ACTION TEST_CASE_2_SETUP:
                        IF vTestCases[1].state = utTestCaseStates.ut_SETUP THEN
	(*Setup the test case information*)
	vTestCases[1].id := 2;
    vTestCases[1].desc[0] := 'RETURNS TRUE WHEN PARAMETER ACT EQUAL TO XP';
    vTestCases[1].desc[1] := 'Tests if the function returns True if the parameter act is equal to parameter xp';
	vTestCases[1].desc[2] := 'PASS IF: Return value is TRUE';
	
	(*Setup needed variables*)
	vTestCase2_act := REAL_TO_LREAL(115.4);
	vTestCase2_xp := REAL_TO_LREAL(115.4);
END_IF
                      
END_ACTION

ACTION TEST_CASE_2_EXEC:
                        IF vTestCases[1].state = utTestCaseStates.ut_RUNNING THEN
	(*Run the test case*)
	IF assertLessEqual_LREAL(vTestCase2_act, vTestCase2_xp) THEN
		vTestCases[1].state := utTestCaseStates.ut_PASSED;
		vTestCases[1].msg := 'Parameter act was equal to xp and function returned TRUE -> PASS';
	ELSE
		vTestCases[1].state := utTestCaseStates.ut_FAILED;
		vTestCases[1].msg := 'Parameter act was equal to xp and function returned FALSE -> FAIL';
	END_IF
END_IF
                      
END_ACTION
END_PROGRAM

PROGRAM test_assertArrayEqual_WORD
  VAR
    vTestCases : ARRAY[0..20] OF utTestCase;  (* Definition of all test cases for this POU *)
    testRunner : utTestSuite;  (* Test Suite fb instance to run the tests *)
    vRunAll : BOOL;  (* Manual command to run all tests for this POU *)
    vResetAll : BOOL;  (* Manual command to reset all tests for this POU *)
    vTestCase1_act : ARRAY[0..70] OF WORD;  (* Array data 1 of test case 1 *)
    vTestCase1_xp : ARRAY[0..70] OF WORD;  (* Array data 2 of test case 1 *)
    vTestCase2_act : ARRAY[0..70] OF WORD;  (* Array data 3 of test case 2 *)
    vTestCase2_xp : ARRAY[0..70] OF WORD;  (* Array data 4 of test case 2 *)
    i : UINT;  (* Iterator variable i *)
    j : UINT;  (* Iterator variable j *)
  END_VAR

                    (*Run the test cases*)
TEST_CASE_1_SETUP();
TEST_CASE_1_EXEC();

TEST_CASE_2_SETUP();
TEST_CASE_2_EXEC();

(*Instantiate the test runner*)
testRunner(
	Id := 140,
	Name := 'assertArrayEqual_WORD',
    RunTests := GVL.RunAll OR vRunAll,
	ResetTests := GVL.ResetAll OR vResetAll,
	TestCases:=vTestCases);

(*Report the results to the collection global*)
GVL.Results[testRunner.Id] := testRunner.Summary;
                  

ACTION TEST_CASE_1_SETUP:
                        IF vTestCases[0].state = utTestCaseStates.ut_SETUP THEN
	(*Setup the test case information*)
	vTestCases[0].id := 1;
	vTestCases[0].desc[0] := 'RETURNS TRUE WHEN ARRAYS EQUAL';
    vTestCases[0].desc[1] := 'Tests if the function returns True if the passed in arrays are identical';
	vTestCases[0].desc[2] := 'PASS IF: Return value is TRUE';
	
	(*Setup needed variables*)
	FOR i:=0 TO 70 DO
		vTestCase1_act[i] := UINT_TO_WORD(35 * BOOL_TO_UINT(i MOD 2 = 0));
		vTestCase1_xp[i] := UINT_TO_WORD(35 * BOOL_TO_UINT(i MOD 2 = 0));
	END_FOR
END_IF
                      
END_ACTION

ACTION TEST_CASE_1_EXEC:
                        IF vTestCases[0].state = utTestCaseStates.ut_RUNNING THEN
	(*Run the test case*)
	IF assertArrayEqual_WORD(ADR(vTestCase1_act), ADR(vTestCase1_xp), SIZEOF(vTestCase1_act)) THEN
		vTestCases[0].state := utTestCaseStates.ut_PASSED;
		vTestCases[0].msg := 'Arrays were equal and function returned TRUE -> PASS';
	ELSE
		vTestCases[0].state := utTestCaseStates.ut_FAILED;
		vTestCases[0].msg := 'Arrays were equal and function returned FALSE -> FAIL';
	END_IF
END_IF
                      
END_ACTION

ACTION TEST_CASE_2_SETUP:
                        IF vTestCases[1].state = utTestCaseStates.ut_SETUP THEN
	(*Setup the test case information*)
	vTestCases[1].id := 2;
	vTestCases[1].desc[0] := 'RETURNS FALSE WHEN ARRAYS NOT EQUAL';
    vTestCases[1].desc[1] := 'Tests if the function returns False if the passed in arrays are not identical';
	vTestCases[1].desc[2] := 'PASS IF: Return value is FALSE';
	
	(*Setup needed variables*)
	FOR j:=0 TO 70 DO
		vTestCase2_act[j] := UINT_TO_WORD(35 * BOOL_TO_UINT(j MOD 2 = 0));
		vTestCase2_xp[j] := UINT_TO_WORD(35 * BOOL_TO_UINT(j MOD 2 <> 0));
	END_FOR
END_IF
                      
END_ACTION

ACTION TEST_CASE_2_EXEC:
                        IF vTestCases[1].state = utTestCaseStates.ut_RUNNING THEN
	(*Run the test case*)
	IF NOT assertArrayEqual_WORD(ADR(vTestCase2_act), ADR(vTestCase2_xp), SIZEOF(vTestCase2_act)) THEN
		vTestCases[1].state := utTestCaseStates.ut_PASSED;
		vTestCases[1].msg := 'Arrays were not equal and function returned FALSE -> PASS';
	ELSE
		vTestCases[1].state := utTestCaseStates.ut_FAILED;
		vTestCases[1].msg := 'Arrays were not equal and function returned TRUE -> FAIL';
	END_IF
END_IF
                      
END_ACTION
END_PROGRAM

PROGRAM test_assertArrayEqual_DWORD
  VAR
    vTestCases : ARRAY[0..20] OF utTestCase;  (* Definition of all test cases for this POU *)
    testRunner : utTestSuite;  (* Test Suite fb instance to run the tests *)
    vRunAll : BOOL;  (* Manual command to run all tests for this POU *)
    vResetAll : BOOL;  (* Manual command to reset all tests for this POU *)
    vTestCase1_act : ARRAY[0..70] OF DWORD;  (* Array data 1 of test case 1 *)
    vTestCase1_xp : ARRAY[0..70] OF DWORD;  (* Array data 2 of test case 1 *)
    vTestCase2_act : ARRAY[0..70] OF DWORD;  (* Array data 3 of test case 2 *)
    vTestCase2_xp : ARRAY[0..70] OF DWORD;  (* Array data 4 of test case 2 *)
    i : UINT;  (* Iterator variable i *)
    j : UINT;  (* Iterator variable j *)
  END_VAR

                    (*Run the test cases*)
TEST_CASE_1_SETUP();
TEST_CASE_1_EXEC();

TEST_CASE_2_SETUP();
TEST_CASE_2_EXEC();

(*Instantiate the test runner*)
testRunner(
	Id := 141,
	Name := 'assertArrayEqual_DWORD',
    RunTests := GVL.RunAll OR vRunAll,
	ResetTests := GVL.ResetAll OR vResetAll,
	TestCases:=vTestCases);

(*Report the results to the collection global*)
GVL.Results[testRunner.Id] := testRunner.Summary;
                  

ACTION TEST_CASE_1_SETUP:
                        IF vTestCases[0].state = utTestCaseStates.ut_SETUP THEN
	(*Setup the test case information*)
	vTestCases[0].id := 1;
	vTestCases[0].desc[0] := 'RETURNS TRUE WHEN ARRAYS EQUAL';
    vTestCases[0].desc[1] := 'Tests if the function returns True if the passed in arrays are identical';
	vTestCases[0].desc[2] := 'PASS IF: Return value is TRUE';
	
	(*Setup needed variables*)
	FOR i:=0 TO 70 DO
		vTestCase1_act[i] := UINT_TO_DWORD(35 * BOOL_TO_UINT(i MOD 2 = 0));
		vTestCase1_xp[i] := UINT_TO_DWORD(35 * BOOL_TO_UINT(i MOD 2 = 0));
	END_FOR
END_IF
                      
END_ACTION

ACTION TEST_CASE_1_EXEC:
                        IF vTestCases[0].state = utTestCaseStates.ut_RUNNING THEN
	(*Run the test case*)
	IF assertArrayEqual_DWORD(ADR(vTestCase1_act), ADR(vTestCase1_xp), SIZEOF(vTestCase1_act)) THEN
		vTestCases[0].state := utTestCaseStates.ut_PASSED;
		vTestCases[0].msg := 'Arrays were equal and function returned TRUE -> PASS';
	ELSE
		vTestCases[0].state := utTestCaseStates.ut_FAILED;
		vTestCases[0].msg := 'Arrays were equal and function returned FALSE -> FAIL';
	END_IF
END_IF
                      
END_ACTION

ACTION TEST_CASE_2_SETUP:
                        IF vTestCases[1].state = utTestCaseStates.ut_SETUP THEN
	(*Setup the test case information*)
	vTestCases[1].id := 2;
	vTestCases[1].desc[0] := 'RETURNS FALSE WHEN ARRAYS NOT EQUAL';
    vTestCases[1].desc[1] := 'Tests if the function returns False if the passed in arrays are not identical';
	vTestCases[1].desc[2] := 'PASS IF: Return value is FALSE';
	
	(*Setup needed variables*)
	FOR j:=0 TO 70 DO
		vTestCase2_act[j] := UINT_TO_DWORD(35 * BOOL_TO_UINT(j MOD 2 = 0));
		vTestCase2_xp[j] := UINT_TO_DWORD(35 * BOOL_TO_UINT(j MOD 2 <> 0));
	END_FOR
END_IF
                      
END_ACTION

ACTION TEST_CASE_2_EXEC:
                        IF vTestCases[1].state = utTestCaseStates.ut_RUNNING THEN
	(*Run the test case*)
	IF NOT assertArrayEqual_DWORD(ADR(vTestCase2_act), ADR(vTestCase2_xp), SIZEOF(vTestCase2_act)) THEN
		vTestCases[1].state := utTestCaseStates.ut_PASSED;
		vTestCases[1].msg := 'Arrays were not equal and function returned FALSE -> PASS';
	ELSE
		vTestCases[1].state := utTestCaseStates.ut_FAILED;
		vTestCases[1].msg := 'Arrays were not equal and function returned TRUE -> FAIL';
	END_IF
END_IF
                      
END_ACTION
END_PROGRAM

PROGRAM test_assertArrayEqual_SINT
  VAR
    vTestCases : ARRAY[0..20] OF utTestCase;  (* Definition of all test cases for this POU *)
    testRunner : utTestSuite;  (* Test Suite fb instance to run the tests *)
    vRunAll : BOOL;  (* Manual command to run all tests for this POU *)
    vResetAll : BOOL;  (* Manual command to reset all tests for this POU *)
    vTestCase1_act : ARRAY[0..70] OF SINT;  (* Array data 1 of test case 1 *)
    vTestCase1_xp : ARRAY[0..70] OF SINT;  (* Array data 2 of test case 1 *)
    vTestCase2_act : ARRAY[0..70] OF SINT;  (* Array data 3 of test case 2 *)
    vTestCase2_xp : ARRAY[0..70] OF SINT;  (* Array data 4 of test case 2 *)
    i : UINT;  (* Iterator variable i *)
    j : UINT;  (* Iterator variable j *)
  END_VAR

                    (*Run the test cases*)
TEST_CASE_1_SETUP();
TEST_CASE_1_EXEC();

TEST_CASE_2_SETUP();
TEST_CASE_2_EXEC();

(*Instantiate the test runner*)
testRunner(
	Id := 143,
	Name := 'assertArrayEqual_SINT',
    RunTests := GVL.RunAll OR vRunAll,
	ResetTests := GVL.ResetAll OR vResetAll,
	TestCases:=vTestCases);

(*Report the results to the collection global*)
GVL.Results[testRunner.Id] := testRunner.Summary;
                  

ACTION TEST_CASE_1_SETUP:
                        IF vTestCases[0].state = utTestCaseStates.ut_SETUP THEN
	(*Setup the test case information*)
	vTestCases[0].id := 1;
	vTestCases[0].desc[0] := 'RETURNS TRUE WHEN ARRAYS EQUAL';
    vTestCases[0].desc[1] := 'Tests if the function returns True if the passed in arrays are identical';
	vTestCases[0].desc[2] := 'PASS IF: Return value is TRUE';
	
	(*Setup needed variables*)
	FOR i:=0 TO 70 DO
		vTestCase1_act[i] := UINT_TO_SINT(35 * BOOL_TO_UINT(i MOD 2 = 0));
		vTestCase1_xp[i] := UINT_TO_SINT(35 * BOOL_TO_UINT(i MOD 2 = 0));
	END_FOR
END_IF
                      
END_ACTION

ACTION TEST_CASE_1_EXEC:
                        IF vTestCases[0].state = utTestCaseStates.ut_RUNNING THEN
	(*Run the test case*)
	IF assertArrayEqual_SINT(ADR(vTestCase1_act), ADR(vTestCase1_xp), SIZEOF(vTestCase1_act)) THEN
		vTestCases[0].state := utTestCaseStates.ut_PASSED;
		vTestCases[0].msg := 'Arrays were equal and function returned TRUE -> PASS';
	ELSE
		vTestCases[0].state := utTestCaseStates.ut_FAILED;
		vTestCases[0].msg := 'Arrays were equal and function returned FALSE -> FAIL';
	END_IF
END_IF
                      
END_ACTION

ACTION TEST_CASE_2_SETUP:
                        IF vTestCases[1].state = utTestCaseStates.ut_SETUP THEN
	(*Setup the test case information*)
	vTestCases[1].id := 2;
	vTestCases[1].desc[0] := 'RETURNS FALSE WHEN ARRAYS NOT EQUAL';
    vTestCases[1].desc[1] := 'Tests if the function returns False if the passed in arrays are not identical';
	vTestCases[1].desc[2] := 'PASS IF: Return value is FALSE';
	
	(*Setup needed variables*)
	FOR j:=0 TO 70 DO
		vTestCase2_act[j] := UINT_TO_SINT(35 * BOOL_TO_UINT(j MOD 2 = 0));
		vTestCase2_xp[j] := UINT_TO_SINT(35 * BOOL_TO_UINT(j MOD 2 <> 0));
	END_FOR
END_IF
                      
END_ACTION

ACTION TEST_CASE_2_EXEC:
                        IF vTestCases[1].state = utTestCaseStates.ut_RUNNING THEN
	(*Run the test case*)
	IF NOT assertArrayEqual_SINT(ADR(vTestCase2_act), ADR(vTestCase2_xp), SIZEOF(vTestCase2_act)) THEN
		vTestCases[1].state := utTestCaseStates.ut_PASSED;
		vTestCases[1].msg := 'Arrays were not equal and function returned FALSE -> PASS';
	ELSE
		vTestCases[1].state := utTestCaseStates.ut_FAILED;
		vTestCases[1].msg := 'Arrays were not equal and function returned TRUE -> FAIL';
	END_IF
END_IF
                      
END_ACTION
END_PROGRAM

PROGRAM test_assertArrayEqual_LREAL
  VAR
    vTestCases : ARRAY[0..20] OF utTestCase;  (* Definition of all test cases for this POU *)
    testRunner : utTestSuite;  (* Test Suite fb instance to run the tests *)
    vRunAll : BOOL;  (* Manual command to run all tests for this POU *)
    vResetAll : BOOL;  (* Manual command to reset all tests for this POU *)
    vTestCase1_act : ARRAY[0..70] OF LREAL;  (* Array data 1 of test case 1 *)
    vTestCase1_xp : ARRAY[0..70] OF LREAL;  (* Array data 2 of test case 1 *)
    vTestCase2_act : ARRAY[0..70] OF LREAL;  (* Array data 3 of test case 2 *)
    vTestCase2_xp : ARRAY[0..70] OF LREAL;  (* Array data 4 of test case 2 *)
    i : UINT;  (* Iterator variable i *)
    j : UINT;  (* Iterator variable j *)
  END_VAR

                    (*Run the test cases*)
TEST_CASE_1_SETUP();
TEST_CASE_1_EXEC();

TEST_CASE_2_SETUP();
TEST_CASE_2_EXEC();

(*Instantiate the test runner*)
testRunner(
	Id := 152,
	Name := 'assertArrayEqual_LREAL',
    RunTests := GVL.RunAll OR vRunAll,
	ResetTests := GVL.ResetAll OR vResetAll,
	TestCases:=vTestCases);

(*Report the results to the collection global*)
GVL.Results[testRunner.Id] := testRunner.Summary;
                  

ACTION TEST_CASE_1_EXEC:
                        IF vTestCases[0].state = utTestCaseStates.ut_RUNNING THEN
	(*Run the test case*)
	IF assertArrayEqual_LREAL(ADR(vTestCase1_act), ADR(vTestCase1_xp), SIZEOF(vTestCase1_act)) THEN
		vTestCases[0].state := utTestCaseStates.ut_PASSED;
		vTestCases[0].msg := 'Arrays were equal and function returned TRUE -> PASS';
	ELSE
		vTestCases[0].state := utTestCaseStates.ut_FAILED;
		vTestCases[0].msg := 'Arrays were equal and function returned FALSE -> FAIL';
	END_IF
END_IF
                      
END_ACTION

ACTION TEST_CASE_2_SETUP:
                        IF vTestCases[1].state = utTestCaseStates.ut_SETUP THEN
	(*Setup the test case information*)
	vTestCases[1].id := 2;
	vTestCases[1].desc[0] := 'RETURNS FALSE WHEN ARRAYS NOT EQUAL';
    vTestCases[1].desc[1] := 'Tests if the function returns False if the passed in arrays are not identical';
	vTestCases[1].desc[2] := 'PASS IF: Return value is FALSE';
	
	(*Setup needed variables*)
	FOR j:=0 TO 70 DO
		vTestCase2_act[j] := UINT_TO_LREAL(35 * BOOL_TO_UINT(j MOD 2 = 0));
		vTestCase2_xp[j] := UINT_TO_LREAL(35 * BOOL_TO_UINT(j MOD 2 <> 0));
	END_FOR
END_IF
                      
END_ACTION

ACTION TEST_CASE_2_EXEC:
                        IF vTestCases[1].state = utTestCaseStates.ut_RUNNING THEN
	(*Run the test case*)
	IF NOT assertArrayEqual_LREAL(ADR(vTestCase2_act), ADR(vTestCase2_xp), SIZEOF(vTestCase2_act)) THEN
		vTestCases[1].state := utTestCaseStates.ut_PASSED;
		vTestCases[1].msg := 'Arrays were not equal and function returned FALSE -> PASS';
	ELSE
		vTestCases[1].state := utTestCaseStates.ut_FAILED;
		vTestCases[1].msg := 'Arrays were not equal and function returned TRUE -> FAIL';
	END_IF
END_IF
                      
END_ACTION

ACTION TEST_CASE_1_SETUP:
                        IF vTestCases[0].state = utTestCaseStates.ut_SETUP THEN
	(*Setup the test case information*)
	vTestCases[0].id := 1;
	vTestCases[0].desc[0] := 'RETURNS TRUE WHEN ARRAYS EQUAL';
    vTestCases[0].desc[1] := 'Tests if the function returns True if the passed in arrays are identical';
	vTestCases[0].desc[2] := 'PASS IF: Return value is TRUE';
	
	(*Setup needed variables*)
	FOR i:=0 TO 70 DO
		vTestCase1_act[i] := UINT_TO_LREAL(35 * BOOL_TO_UINT(i MOD 2 = 0));
		vTestCase1_xp[i] := UINT_TO_LREAL(35 * BOOL_TO_UINT(i MOD 2 = 0));
	END_FOR
END_IF
                      
END_ACTION
END_PROGRAM

PROGRAM test_assertLessEqual_LTIME
  VAR
    vTestCases : ARRAY[0..20] OF utTestCase;  (* Definition of all test cases for this POU *)
    testRunner : utTestSuite;  (* Test Suite fb instance to run the tests *)
    vRunAll : BOOL;  (* Manual command to run all tests for this POU *)
    vResetAll : BOOL;  (* Manual command to reset all tests for this POU *)
    vTestCase1_act : LTIME;  (* Test data 1 of test case 1 *)
    vTestCase1_xp : LTIME;  (* Test data 2 of test case 1 *)
    vTestCase2_act : LTIME;  (* Test data 1 of test case 2 *)
    vTestCase2_xp : LTIME;  (* Test data 2 of test case 2 *)
    vTestCase3_act : LTIME;  (* Test data 1 of test case 3 *)
    vTestCase3_xp : LTIME;  (* Test data 2 of test case 3 *)
  END_VAR

                    (*Run the test cases*)
TEST_CASE_1_SETUP();
TEST_CASE_1_EXEC();

TEST_CASE_2_SETUP();
TEST_CASE_2_EXEC();

TEST_CASE_3_SETUP();
TEST_CASE_3_EXEC();

(*Instantiate the test runner*)
testRunner(
	Id := 131,
	Name := 'assertLessEqual_LTIME',
    RunTests := GVL.RunAll OR vRunAll,
	ResetTests := GVL.ResetAll OR vResetAll,
	TestCases:=vTestCases);

(*Report the results to the collection global*)
GVL.Results[testRunner.Id] := testRunner.Summary;
                  

ACTION TEST_CASE_1_EXEC:
                        IF vTestCases[0].state = utTestCaseStates.ut_RUNNING THEN
	(*Run the test case*)
	IF assertLessEqual_LTIME(vTestCase1_act, vTestCase1_xp) THEN
		vTestCases[0].state := utTestCaseStates.ut_PASSED;
		vTestCases[0].msg := 'Parameter act was less than xp and function returned TRUE -> PASS';
	ELSE
		vTestCases[0].state := utTestCaseStates.ut_FAILED;
		vTestCases[0].msg := 'Parameter act was less than xp and function returned FALSE -> FAIL';
	END_IF
END_IF
                      
END_ACTION

ACTION TEST_CASE_3_SETUP:
                        IF vTestCases[2].state = utTestCaseStates.ut_SETUP THEN
	(*Setup the test case information*)
	vTestCases[2].id := 3;
    vTestCases[2].desc[0] := 'RETURNS FALSE WHEN PARAMETER ACT GREATER THAN XP';
    vTestCases[2].desc[1] := 'Tests if the function returns False if the parameter act is greater than parameter xp';
	vTestCases[2].desc[2] := 'PASS IF: Return value is FALSE';
	
	(*Setup needed variables*)
	vTestCase3_act := REAL_TO_LTIME(115.4);
	vTestCase3_xp := REAL_TO_LTIME(85.4);
END_IF
                      
END_ACTION

ACTION TEST_CASE_3_EXEC:
                        IF vTestCases[2].state = utTestCaseStates.ut_RUNNING THEN
	(*Run the test case*)
	IF NOT assertLessEqual_LTIME(vTestCase3_act, vTestCase3_xp) THEN
		vTestCases[2].state := utTestCaseStates.ut_PASSED;
		vTestCases[2].msg := 'Parameter act was greater than xp and function returned FALSE -> PASS';
	ELSE
		vTestCases[2].state := utTestCaseStates.ut_FAILED;
		vTestCases[2].msg := 'Parameter act was greater than xp and function returned TRUE -> FAIL';
	END_IF
END_IF
                      
END_ACTION

ACTION TEST_CASE_1_SETUP:
                        IF vTestCases[0].state = utTestCaseStates.ut_SETUP THEN
	(*Setup the test case information*)
	vTestCases[0].id := 1;
	vTestCases[0].desc[0] := 'RETURNS TRUE WHEN PARAMETER ACT LESS THAN XP';
    vTestCases[0].desc[1] := 'Tests if the function returns True if the parameter act is less than parameter xp';
	vTestCases[0].desc[2] := 'PASS IF: Return value is TRUE';
	
	(*Setup needed variables*)
	vTestCase1_act := REAL_TO_LTIME(85.4);
	vTestCase1_xp := REAL_TO_LTIME(115.4);
END_IF
                      
END_ACTION

ACTION TEST_CASE_2_SETUP:
                        IF vTestCases[1].state = utTestCaseStates.ut_SETUP THEN
	(*Setup the test case information*)
	vTestCases[1].id := 2;
    vTestCases[1].desc[0] := 'RETURNS TRUE WHEN PARAMETER ACT EQUAL TO XP';
    vTestCases[1].desc[1] := 'Tests if the function returns True if the parameter act is equal to parameter xp';
	vTestCases[1].desc[2] := 'PASS IF: Return value is TRUE';
	
	(*Setup needed variables*)
	vTestCase2_act := REAL_TO_LTIME(115.4);
	vTestCase2_xp := REAL_TO_LTIME(115.4);
END_IF
                      
END_ACTION

ACTION TEST_CASE_2_EXEC:
                        IF vTestCases[1].state = utTestCaseStates.ut_RUNNING THEN
	(*Run the test case*)
	IF assertLessEqual_LTIME(vTestCase2_act, vTestCase2_xp) THEN
		vTestCases[1].state := utTestCaseStates.ut_PASSED;
		vTestCases[1].msg := 'Parameter act was equal to xp and function returned TRUE -> PASS';
	ELSE
		vTestCases[1].state := utTestCaseStates.ut_FAILED;
		vTestCases[1].msg := 'Parameter act was equal to xp and function returned FALSE -> FAIL';
	END_IF
END_IF
                      
END_ACTION
END_PROGRAM

PROGRAM test_assertArrayEqual_LINT
  VAR
    vTestCases : ARRAY[0..20] OF utTestCase;  (* Definition of all test cases for this POU *)
    testRunner : utTestSuite;  (* Test Suite fb instance to run the tests *)
    vRunAll : BOOL;  (* Manual command to run all tests for this POU *)
    vResetAll : BOOL;  (* Manual command to reset all tests for this POU *)
    vTestCase1_act : ARRAY[0..70] OF LINT;  (* Array data 1 of test case 1 *)
    vTestCase1_xp : ARRAY[0..70] OF LINT;  (* Array data 2 of test case 1 *)
    vTestCase2_act : ARRAY[0..70] OF LINT;  (* Array data 3 of test case 2 *)
    vTestCase2_xp : ARRAY[0..70] OF LINT;  (* Array data 4 of test case 2 *)
    i : UINT;  (* Iterator variable i *)
    j : UINT;  (* Iterator variable j *)
  END_VAR

                    (*Run the test cases*)
TEST_CASE_1_SETUP();
TEST_CASE_1_EXEC();

TEST_CASE_2_SETUP();
TEST_CASE_2_EXEC();

(*Instantiate the test runner*)
testRunner(
	Id := 149,
	Name := 'assertArrayEqual_LINT',
    RunTests := GVL.RunAll OR vRunAll,
	ResetTests := GVL.ResetAll OR vResetAll,
	TestCases:=vTestCases);

(*Report the results to the collection global*)
GVL.Results[testRunner.Id] := testRunner.Summary;
                  

ACTION TEST_CASE_2_SETUP:
                        IF vTestCases[1].state = utTestCaseStates.ut_SETUP THEN
	(*Setup the test case information*)
	vTestCases[1].id := 2;
	vTestCases[1].desc[0] := 'RETURNS FALSE WHEN ARRAYS NOT EQUAL';
    vTestCases[1].desc[1] := 'Tests if the function returns False if the passed in arrays are not identical';
	vTestCases[1].desc[2] := 'PASS IF: Return value is FALSE';
	
	(*Setup needed variables*)
	FOR j:=0 TO 70 DO
		vTestCase2_act[j] := UINT_TO_LINT(35 * BOOL_TO_UINT(j MOD 2 = 0));
		vTestCase2_xp[j] := UINT_TO_LINT(35 * BOOL_TO_UINT(j MOD 2 <> 0));
	END_FOR
END_IF
                      
END_ACTION

ACTION TEST_CASE_1_SETUP:
                        IF vTestCases[0].state = utTestCaseStates.ut_SETUP THEN
	(*Setup the test case information*)
	vTestCases[0].id := 1;
	vTestCases[0].desc[0] := 'RETURNS TRUE WHEN ARRAYS EQUAL';
    vTestCases[0].desc[1] := 'Tests if the function returns True if the passed in arrays are identical';
	vTestCases[0].desc[2] := 'PASS IF: Return value is TRUE';
	
	(*Setup needed variables*)
	FOR i:=0 TO 70 DO
		vTestCase1_act[i] := UINT_TO_LINT(35 * BOOL_TO_UINT(i MOD 2 = 0));
		vTestCase1_xp[i] := UINT_TO_LINT(35 * BOOL_TO_UINT(i MOD 2 = 0));
	END_FOR
END_IF
                      
END_ACTION

ACTION TEST_CASE_1_EXEC:
                        IF vTestCases[0].state = utTestCaseStates.ut_RUNNING THEN
	(*Run the test case*)
	IF assertArrayEqual_LINT(ADR(vTestCase1_act), ADR(vTestCase1_xp), SIZEOF(vTestCase1_act)) THEN
		vTestCases[0].state := utTestCaseStates.ut_PASSED;
		vTestCases[0].msg := 'Arrays were equal and function returned TRUE -> PASS';
	ELSE
		vTestCases[0].state := utTestCaseStates.ut_FAILED;
		vTestCases[0].msg := 'Arrays were equal and function returned FALSE -> FAIL';
	END_IF
END_IF
                      
END_ACTION

ACTION TEST_CASE_2_EXEC:
                        IF vTestCases[1].state = utTestCaseStates.ut_RUNNING THEN
	(*Run the test case*)
	IF NOT assertArrayEqual_LINT(ADR(vTestCase2_act), ADR(vTestCase2_xp), SIZEOF(vTestCase2_act)) THEN
		vTestCases[1].state := utTestCaseStates.ut_PASSED;
		vTestCases[1].msg := 'Arrays were not equal and function returned FALSE -> PASS';
	ELSE
		vTestCases[1].state := utTestCaseStates.ut_FAILED;
		vTestCases[1].msg := 'Arrays were not equal and function returned TRUE -> FAIL';
	END_IF
END_IF
                      
END_ACTION
END_PROGRAM

PROGRAM test_assertLessEqual_REAL
  VAR
    vTestCases : ARRAY[0..20] OF utTestCase;  (* Definition of all test cases for this POU *)
    testRunner : utTestSuite;  (* Test Suite fb instance to run the tests *)
    vRunAll : BOOL;  (* Manual command to run all tests for this POU *)
    vResetAll : BOOL;  (* Manual command to reset all tests for this POU *)
    vTestCase1_act : REAL;  (* Test data 1 of test case 1 *)
    vTestCase1_xp : REAL;  (* Test data 2 of test case 1 *)
    vTestCase2_act : REAL;  (* Test data 1 of test case 2 *)
    vTestCase2_xp : REAL;  (* Test data 2 of test case 2 *)
    vTestCase3_act : REAL;  (* Test data 1 of test case 3 *)
    vTestCase3_xp : REAL;  (* Test data 2 of test case 3 *)
  END_VAR

                    (*Run the test cases*)
TEST_CASE_1_SETUP();
TEST_CASE_1_EXEC();

TEST_CASE_2_SETUP();
TEST_CASE_2_EXEC();

TEST_CASE_3_SETUP();
TEST_CASE_3_EXEC();

(*Instantiate the test runner*)
testRunner(
	Id := 128,
	Name := 'assertLessEqual_REAL',
    RunTests := GVL.RunAll OR vRunAll,
	ResetTests := GVL.ResetAll OR vResetAll,
	TestCases:=vTestCases);

(*Report the results to the collection global*)
GVL.Results[testRunner.Id] := testRunner.Summary;
                  

ACTION TEST_CASE_2_SETUP:
                        IF vTestCases[1].state = utTestCaseStates.ut_SETUP THEN
	(*Setup the test case information*)
	vTestCases[1].id := 2;
    vTestCases[1].desc[0] := 'RETURNS TRUE WHEN PARAMETER ACT EQUAL TO XP';
    vTestCases[1].desc[1] := 'Tests if the function returns True if the parameter act is equal to parameter xp';
	vTestCases[1].desc[2] := 'PASS IF: Return value is TRUE';
	
	(*Setup needed variables*)
	vTestCase2_act := 115.4;
	vTestCase2_xp := 115.4;
END_IF
                      
END_ACTION

ACTION TEST_CASE_3_SETUP:
                        IF vTestCases[2].state = utTestCaseStates.ut_SETUP THEN
	(*Setup the test case information*)
	vTestCases[2].id := 3;
    vTestCases[2].desc[0] := 'RETURNS FALSE WHEN PARAMETER ACT GREATER THAN XP';
    vTestCases[2].desc[1] := 'Tests if the function returns False if the parameter act is greater than parameter xp';
	vTestCases[2].desc[2] := 'PASS IF: Return value is FALSE';
	
	(*Setup needed variables*)
	vTestCase3_act := 115.4;
	vTestCase3_xp := 85.4;
END_IF
                      
END_ACTION

ACTION TEST_CASE_3_EXEC:
                        IF vTestCases[2].state = utTestCaseStates.ut_RUNNING THEN
	(*Run the test case*)
	IF NOT assertLessEqual_REAL(vTestCase3_act, vTestCase3_xp) THEN
		vTestCases[2].state := utTestCaseStates.ut_PASSED;
		vTestCases[2].msg := 'Parameter act was greater than xp and function returned FALSE -> PASS';
	ELSE
		vTestCases[2].state := utTestCaseStates.ut_FAILED;
		vTestCases[2].msg := 'Parameter act was greater than xp and function returned TRUE -> FAIL';
	END_IF
END_IF
                      
END_ACTION

ACTION TEST_CASE_2_EXEC:
                        IF vTestCases[1].state = utTestCaseStates.ut_RUNNING THEN
	(*Run the test case*)
	IF assertLessEqual_REAL(vTestCase2_act, vTestCase2_xp) THEN
		vTestCases[1].state := utTestCaseStates.ut_PASSED;
		vTestCases[1].msg := 'Parameter act was equal to xp and function returned TRUE -> PASS';
	ELSE
		vTestCases[1].state := utTestCaseStates.ut_FAILED;
		vTestCases[1].msg := 'Parameter act was equal to xp and function returned FALSE -> FAIL';
	END_IF
END_IF
                      
END_ACTION

ACTION TEST_CASE_1_SETUP:
                        IF vTestCases[0].state = utTestCaseStates.ut_SETUP THEN
	(*Setup the test case information*)
	vTestCases[0].id := 1;
	vTestCases[0].desc[0] := 'RETURNS TRUE WHEN PARAMETER ACT LESS THAN XP';
    vTestCases[0].desc[1] := 'Tests if the function returns True if the parameter act is less than parameter xp';
	vTestCases[0].desc[2] := 'PASS IF: Return value is TRUE';
	
	(*Setup needed variables*)
	vTestCase1_act := 85.4;
	vTestCase1_xp := 115.4;
END_IF
                      
END_ACTION

ACTION TEST_CASE_1_EXEC:
                        IF vTestCases[0].state = utTestCaseStates.ut_RUNNING THEN
	(*Run the test case*)
	IF assertLessEqual_REAL(vTestCase1_act, vTestCase1_xp) THEN
		vTestCases[0].state := utTestCaseStates.ut_PASSED;
		vTestCases[0].msg := 'Parameter act was less than xp and function returned TRUE -> PASS';
	ELSE
		vTestCases[0].state := utTestCaseStates.ut_FAILED;
		vTestCases[0].msg := 'Parameter act was less than xp and function returned FALSE -> FAIL';
	END_IF
END_IF
                      
END_ACTION
END_PROGRAM

PROGRAM test_assertArrayEqual_DINT
  VAR
    vTestCases : ARRAY[0..20] OF utTestCase;  (* Definition of all test cases for this POU *)
    testRunner : utTestSuite;  (* Test Suite fb instance to run the tests *)
    vRunAll : BOOL;  (* Manual command to run all tests for this POU *)
    vResetAll : BOOL;  (* Manual command to reset all tests for this POU *)
    vTestCase1_act : ARRAY[0..70] OF DINT;  (* Array data 1 of test case 1 *)
    vTestCase1_xp : ARRAY[0..70] OF DINT;  (* Array data 2 of test case 1 *)
    vTestCase2_act : ARRAY[0..70] OF DINT;  (* Array data 3 of test case 2 *)
    vTestCase2_xp : ARRAY[0..70] OF DINT;  (* Array data 4 of test case 2 *)
    i : UINT;  (* Iterator variable i *)
    j : UINT;  (* Iterator variable j *)
  END_VAR

                    (*Run the test cases*)
TEST_CASE_1_SETUP();
TEST_CASE_1_EXEC();

TEST_CASE_2_SETUP();
TEST_CASE_2_EXEC();

(*Instantiate the test runner*)
testRunner(
	Id := 147,
	Name := 'assertArrayEqual_DINT',
    RunTests := GVL.RunAll OR vRunAll,
	ResetTests := GVL.ResetAll OR vResetAll,
	TestCases:=vTestCases);

(*Report the results to the collection global*)
GVL.Results[testRunner.Id] := testRunner.Summary;
                  

ACTION TEST_CASE_1_SETUP:
                        IF vTestCases[0].state = utTestCaseStates.ut_SETUP THEN
	(*Setup the test case information*)
	vTestCases[0].id := 1;
	vTestCases[0].desc[0] := 'RETURNS TRUE WHEN ARRAYS EQUAL';
    vTestCases[0].desc[1] := 'Tests if the function returns True if the passed in arrays are identical';
	vTestCases[0].desc[2] := 'PASS IF: Return value is TRUE';
	
	(*Setup needed variables*)
	FOR i:=0 TO 70 DO
		vTestCase1_act[i] := UINT_TO_DINT(35 * BOOL_TO_UINT(i MOD 2 = 0));
		vTestCase1_xp[i] := UINT_TO_DINT(35 * BOOL_TO_UINT(i MOD 2 = 0));
	END_FOR
END_IF
                      
END_ACTION

ACTION TEST_CASE_1_EXEC:
                        IF vTestCases[0].state = utTestCaseStates.ut_RUNNING THEN
	(*Run the test case*)
	IF assertArrayEqual_DINT(ADR(vTestCase1_act), ADR(vTestCase1_xp), SIZEOF(vTestCase1_act)) THEN
		vTestCases[0].state := utTestCaseStates.ut_PASSED;
		vTestCases[0].msg := 'Arrays were equal and function returned TRUE -> PASS';
	ELSE
		vTestCases[0].state := utTestCaseStates.ut_FAILED;
		vTestCases[0].msg := 'Arrays were equal and function returned FALSE -> FAIL';
	END_IF
END_IF
                      
END_ACTION

ACTION TEST_CASE_2_SETUP:
                        IF vTestCases[1].state = utTestCaseStates.ut_SETUP THEN
	(*Setup the test case information*)
	vTestCases[1].id := 2;
	vTestCases[1].desc[0] := 'RETURNS FALSE WHEN ARRAYS NOT EQUAL';
    vTestCases[1].desc[1] := 'Tests if the function returns False if the passed in arrays are not identical';
	vTestCases[1].desc[2] := 'PASS IF: Return value is FALSE';
	
	(*Setup needed variables*)
	FOR j:=0 TO 70 DO
		vTestCase2_act[j] := UINT_TO_DINT(35 * BOOL_TO_UINT(j MOD 2 = 0));
		vTestCase2_xp[j] := UINT_TO_DINT(35 * BOOL_TO_UINT(j MOD 2 <> 0));
	END_FOR
END_IF
                      
END_ACTION

ACTION TEST_CASE_2_EXEC:
                        IF vTestCases[1].state = utTestCaseStates.ut_RUNNING THEN
	(*Run the test case*)
	IF NOT assertArrayEqual_DINT(ADR(vTestCase2_act), ADR(vTestCase2_xp), SIZEOF(vTestCase2_act)) THEN
		vTestCases[1].state := utTestCaseStates.ut_PASSED;
		vTestCases[1].msg := 'Arrays were not equal and function returned FALSE -> PASS';
	ELSE
		vTestCases[1].state := utTestCaseStates.ut_FAILED;
		vTestCases[1].msg := 'Arrays were not equal and function returned TRUE -> FAIL';
	END_IF
END_IF
                      
END_ACTION
END_PROGRAM

PROGRAM test_assertArrayEqual_UDINT
  VAR
    vTestCases : ARRAY[0..20] OF utTestCase;  (* Definition of all test cases for this POU *)
    testRunner : utTestSuite;  (* Test Suite fb instance to run the tests *)
    vRunAll : BOOL;  (* Manual command to run all tests for this POU *)
    vResetAll : BOOL;  (* Manual command to reset all tests for this POU *)
    vTestCase1_act : ARRAY[0..70] OF UDINT;  (* Array data 1 of test case 1 *)
    vTestCase1_xp : ARRAY[0..70] OF UDINT;  (* Array data 2 of test case 1 *)
    vTestCase2_act : ARRAY[0..70] OF UDINT;  (* Array data 3 of test case 2 *)
    vTestCase2_xp : ARRAY[0..70] OF UDINT;  (* Array data 4 of test case 2 *)
    i : UINT;  (* Iterator variable i *)
    j : UINT;  (* Iterator variable j *)
  END_VAR

                    (*Run the test cases*)
TEST_CASE_1_SETUP();
TEST_CASE_1_EXEC();

TEST_CASE_2_SETUP();
TEST_CASE_2_EXEC();

(*Instantiate the test runner*)
testRunner(
	Id := 148,
	Name := 'assertArrayEqual_UDINT',
    RunTests := GVL.RunAll OR vRunAll,
	ResetTests := GVL.ResetAll OR vResetAll,
	TestCases:=vTestCases);

(*Report the results to the collection global*)
GVL.Results[testRunner.Id] := testRunner.Summary;
                  

ACTION TEST_CASE_1_SETUP:
                        IF vTestCases[0].state = utTestCaseStates.ut_SETUP THEN
	(*Setup the test case information*)
	vTestCases[0].id := 1;
	vTestCases[0].desc[0] := 'RETURNS TRUE WHEN ARRAYS EQUAL';
    vTestCases[0].desc[1] := 'Tests if the function returns True if the passed in arrays are identical';
	vTestCases[0].desc[2] := 'PASS IF: Return value is TRUE';
	
	(*Setup needed variables*)
	FOR i:=0 TO 70 DO
		vTestCase1_act[i] := UINT_TO_UDINT(35 * BOOL_TO_UINT(i MOD 2 = 0));
		vTestCase1_xp[i] := UINT_TO_UDINT(35 * BOOL_TO_UINT(i MOD 2 = 0));
	END_FOR
END_IF
                      
END_ACTION

ACTION TEST_CASE_1_EXEC:
                        IF vTestCases[0].state = utTestCaseStates.ut_RUNNING THEN
	(*Run the test case*)
	IF assertArrayEqual_UDINT(ADR(vTestCase1_act), ADR(vTestCase1_xp), SIZEOF(vTestCase1_act)) THEN
		vTestCases[0].state := utTestCaseStates.ut_PASSED;
		vTestCases[0].msg := 'Arrays were equal and function returned TRUE -> PASS';
	ELSE
		vTestCases[0].state := utTestCaseStates.ut_FAILED;
		vTestCases[0].msg := 'Arrays were equal and function returned FALSE -> FAIL';
	END_IF
END_IF
                      
END_ACTION

ACTION TEST_CASE_2_SETUP:
                        IF vTestCases[1].state = utTestCaseStates.ut_SETUP THEN
	(*Setup the test case information*)
	vTestCases[1].id := 2;
	vTestCases[1].desc[0] := 'RETURNS FALSE WHEN ARRAYS NOT EQUAL';
    vTestCases[1].desc[1] := 'Tests if the function returns False if the passed in arrays are not identical';
	vTestCases[1].desc[2] := 'PASS IF: Return value is FALSE';
	
	(*Setup needed variables*)
	FOR j:=0 TO 70 DO
		vTestCase2_act[j] := UINT_TO_UDINT(35 * BOOL_TO_UINT(j MOD 2 = 0));
		vTestCase2_xp[j] := UINT_TO_UDINT(35 * BOOL_TO_UINT(j MOD 2 <> 0));
	END_FOR
END_IF
                      
END_ACTION

ACTION TEST_CASE_2_EXEC:
                        IF vTestCases[1].state = utTestCaseStates.ut_RUNNING THEN
	(*Run the test case*)
	IF NOT assertArrayEqual_UDINT(ADR(vTestCase2_act), ADR(vTestCase2_xp), SIZEOF(vTestCase2_act)) THEN
		vTestCases[1].state := utTestCaseStates.ut_PASSED;
		vTestCases[1].msg := 'Arrays were not equal and function returned FALSE -> PASS';
	ELSE
		vTestCases[1].state := utTestCaseStates.ut_FAILED;
		vTestCases[1].msg := 'Arrays were not equal and function returned TRUE -> FAIL';
	END_IF
END_IF
                      
END_ACTION
END_PROGRAM

PROGRAM test_assertLessEqual_LDATE_AND_TIME
  VAR
    vTestCases : ARRAY[0..20] OF utTestCase;  (* Definition of all test cases for this POU *)
    testRunner : utTestSuite;  (* Test Suite fb instance to run the tests *)
    vRunAll : BOOL;  (* Manual command to run all tests for this POU *)
    vResetAll : BOOL;  (* Manual command to reset all tests for this POU *)
    vTestCase1_act : LDATE_AND_TIME;  (* Test data 1 of test case 1 *)
    vTestCase1_xp : LDATE_AND_TIME;  (* Test data 2 of test case 1 *)
    vTestCase2_act : LDATE_AND_TIME;  (* Test data 1 of test case 2 *)
    vTestCase2_xp : LDATE_AND_TIME;  (* Test data 2 of test case 2 *)
    vTestCase3_act : LDATE_AND_TIME;  (* Test data 1 of test case 3 *)
    vTestCase3_xp : LDATE_AND_TIME;  (* Test data 2 of test case 3 *)
  END_VAR

                    (*Run the test cases*)
TEST_CASE_1_SETUP();
TEST_CASE_1_EXEC();

TEST_CASE_2_SETUP();
TEST_CASE_2_EXEC();

TEST_CASE_3_SETUP();
TEST_CASE_3_EXEC();

(*Instantiate the test runner*)
testRunner(
	Id := 135,
	Name := 'assertLessEqual_LDATE_AND_TIME',
    RunTests := GVL.RunAll OR vRunAll,
	ResetTests := GVL.ResetAll OR vResetAll,
	TestCases:=vTestCases);

(*Report the results to the collection global*)
GVL.Results[testRunner.Id] := testRunner.Summary;
                  

ACTION TEST_CASE_2_SETUP:
                        IF vTestCases[1].state = utTestCaseStates.ut_SETUP THEN
	(*Setup the test case information*)
	vTestCases[1].id := 2;
    vTestCases[1].desc[0] := 'RETURNS TRUE WHEN PARAMETER ACT EQUAL TO XP';
    vTestCases[1].desc[1] := 'Tests if the function returns True if the parameter act is equal to parameter xp';
	vTestCases[1].desc[2] := 'PASS IF: Return value is TRUE';
	
	(*Setup needed variables*)
	vTestCase2_act := REAL_TO_LDT(115.4);
	vTestCase2_xp := REAL_TO_LDT(115.4);
END_IF
                      
END_ACTION

ACTION TEST_CASE_3_SETUP:
                        IF vTestCases[2].state = utTestCaseStates.ut_SETUP THEN
	(*Setup the test case information*)
	vTestCases[2].id := 3;
    vTestCases[2].desc[0] := 'RETURNS FALSE WHEN PARAMETER ACT GREATER THAN XP';
    vTestCases[2].desc[1] := 'Tests if the function returns False if the parameter act is greater than parameter xp';
	vTestCases[2].desc[2] := 'PASS IF: Return value is FALSE';
	
	(*Setup needed variables*)
	vTestCase3_act := REAL_TO_LDT(115.4);
	vTestCase3_xp := REAL_TO_LDT(85.4);
END_IF
                      
END_ACTION

ACTION TEST_CASE_3_EXEC:
                        IF vTestCases[2].state = utTestCaseStates.ut_RUNNING THEN
	(*Run the test case*)
	IF NOT assertLessEqual_LDATE_AND_TIME(vTestCase3_act, vTestCase3_xp) THEN
		vTestCases[2].state := utTestCaseStates.ut_PASSED;
		vTestCases[2].msg := 'Parameter act was greater than xp and function returned FALSE -> PASS';
	ELSE
		vTestCases[2].state := utTestCaseStates.ut_FAILED;
		vTestCases[2].msg := 'Parameter act was greater than xp and function returned TRUE -> FAIL';
	END_IF
END_IF
                      
END_ACTION

ACTION TEST_CASE_1_SETUP:
                        IF vTestCases[0].state = utTestCaseStates.ut_SETUP THEN
	(*Setup the test case information*)
	vTestCases[0].id := 1;
	vTestCases[0].desc[0] := 'RETURNS TRUE WHEN PARAMETER ACT LESS THAN XP';
    vTestCases[0].desc[1] := 'Tests if the function returns True if the parameter act is less than parameter xp';
	vTestCases[0].desc[2] := 'PASS IF: Return value is TRUE';
	
	(*Setup needed variables*)
	vTestCase1_act := REAL_TO_LDT(85.4);
	vTestCase1_xp := REAL_TO_LDT(115.4);
END_IF
                      
END_ACTION

ACTION TEST_CASE_1_EXEC:
                        IF vTestCases[0].state = utTestCaseStates.ut_RUNNING THEN
	(*Run the test case*)
	IF assertLessEqual_LDATE_AND_TIME(vTestCase1_act, vTestCase1_xp) THEN
		vTestCases[0].state := utTestCaseStates.ut_PASSED;
		vTestCases[0].msg := 'Parameter act was less than xp and function returned TRUE -> PASS';
	ELSE
		vTestCases[0].state := utTestCaseStates.ut_FAILED;
		vTestCases[0].msg := 'Parameter act was less than xp and function returned FALSE -> FAIL';
	END_IF
END_IF
                      
END_ACTION

ACTION TEST_CASE_2_EXEC:
                        IF vTestCases[1].state = utTestCaseStates.ut_RUNNING THEN
	(*Run the test case*)
	IF assertLessEqual_LDATE_AND_TIME(vTestCase2_act, vTestCase2_xp) THEN
		vTestCases[1].state := utTestCaseStates.ut_PASSED;
		vTestCases[1].msg := 'Parameter act was equal to xp and function returned TRUE -> PASS';
	ELSE
		vTestCases[1].state := utTestCaseStates.ut_FAILED;
		vTestCases[1].msg := 'Parameter act was equal to xp and function returned FALSE -> FAIL';
	END_IF
END_IF
                      
END_ACTION
END_PROGRAM

PROGRAM test_assertArrayEqual_ULINT
  VAR
    vTestCases : ARRAY[0..20] OF utTestCase;  (* Definition of all test cases for this POU *)
    testRunner : utTestSuite;  (* Test Suite fb instance to run the tests *)
    vRunAll : BOOL;  (* Manual command to run all tests for this POU *)
    vResetAll : BOOL;  (* Manual command to reset all tests for this POU *)
    vTestCase1_act : ARRAY[0..70] OF ULINT;  (* Array data 1 of test case 1 *)
    vTestCase1_xp : ARRAY[0..70] OF ULINT;  (* Array data 2 of test case 1 *)
    vTestCase2_act : ARRAY[0..70] OF ULINT;  (* Array data 3 of test case 2 *)
    vTestCase2_xp : ARRAY[0..70] OF ULINT;  (* Array data 4 of test case 2 *)
    i : UINT;  (* Iterator variable i *)
    j : UINT;  (* Iterator variable j *)
  END_VAR

                    (*Run the test cases*)
TEST_CASE_1_SETUP();
TEST_CASE_1_EXEC();

TEST_CASE_2_SETUP();
TEST_CASE_2_EXEC();

(*Instantiate the test runner*)
testRunner(
	Id := 150,
	Name := 'assertArrayEqual_ULINT',
    RunTests := GVL.RunAll OR vRunAll,
	ResetTests := GVL.ResetAll OR vResetAll,
	TestCases:=vTestCases);

(*Report the results to the collection global*)
GVL.Results[testRunner.Id] := testRunner.Summary;
                  

ACTION TEST_CASE_1_SETUP:
                        IF vTestCases[0].state = utTestCaseStates.ut_SETUP THEN
	(*Setup the test case information*)
	vTestCases[0].id := 1;
	vTestCases[0].desc[0] := 'RETURNS TRUE WHEN ARRAYS EQUAL';
    vTestCases[0].desc[1] := 'Tests if the function returns True if the passed in arrays are identical';
	vTestCases[0].desc[2] := 'PASS IF: Return value is TRUE';
	
	(*Setup needed variables*)
	FOR i:=0 TO 70 DO
		vTestCase1_act[i] := UINT_TO_ULINT(35 * BOOL_TO_UINT(i MOD 2 = 0));
		vTestCase1_xp[i] := UINT_TO_ULINT(35 * BOOL_TO_UINT(i MOD 2 = 0));
	END_FOR
END_IF
                      
END_ACTION

ACTION TEST_CASE_1_EXEC:
                        IF vTestCases[0].state = utTestCaseStates.ut_RUNNING THEN
	(*Run the test case*)
	IF assertArrayEqual_ULINT(ADR(vTestCase1_act), ADR(vTestCase1_xp), SIZEOF(vTestCase1_act)) THEN
		vTestCases[0].state := utTestCaseStates.ut_PASSED;
		vTestCases[0].msg := 'Arrays were equal and function returned TRUE -> PASS';
	ELSE
		vTestCases[0].state := utTestCaseStates.ut_FAILED;
		vTestCases[0].msg := 'Arrays were equal and function returned FALSE -> FAIL';
	END_IF
END_IF
                      
END_ACTION

ACTION TEST_CASE_2_SETUP:
                        IF vTestCases[1].state = utTestCaseStates.ut_SETUP THEN
	(*Setup the test case information*)
	vTestCases[1].id := 2;
	vTestCases[1].desc[0] := 'RETURNS FALSE WHEN ARRAYS NOT EQUAL';
    vTestCases[1].desc[1] := 'Tests if the function returns False if the passed in arrays are not identical';
	vTestCases[1].desc[2] := 'PASS IF: Return value is FALSE';
	
	(*Setup needed variables*)
	FOR j:=0 TO 70 DO
		vTestCase2_act[j] := UINT_TO_ULINT(35 * BOOL_TO_UINT(j MOD 2 = 0));
		vTestCase2_xp[j] := UINT_TO_ULINT(35 * BOOL_TO_UINT(j MOD 2 <> 0));
	END_FOR
END_IF
                      
END_ACTION

ACTION TEST_CASE_2_EXEC:
                        IF vTestCases[1].state = utTestCaseStates.ut_RUNNING THEN
	(*Run the test case*)
	IF NOT assertArrayEqual_ULINT(ADR(vTestCase2_act), ADR(vTestCase2_xp), SIZEOF(vTestCase2_act)) THEN
		vTestCases[1].state := utTestCaseStates.ut_PASSED;
		vTestCases[1].msg := 'Arrays were not equal and function returned FALSE -> PASS';
	ELSE
		vTestCases[1].state := utTestCaseStates.ut_FAILED;
		vTestCases[1].msg := 'Arrays were not equal and function returned TRUE -> FAIL';
	END_IF
END_IF
                      
END_ACTION
END_PROGRAM

PROGRAM test_assertArrayEqual_LWORD
  VAR
    vTestCases : ARRAY[0..20] OF utTestCase;  (* Definition of all test cases for this POU *)
    testRunner : utTestSuite;  (* Test Suite fb instance to run the tests *)
    vRunAll : BOOL;  (* Manual command to run all tests for this POU *)
    vResetAll : BOOL;  (* Manual command to reset all tests for this POU *)
    vTestCase1_act : ARRAY[0..70] OF LWORD;  (* Array data 1 of test case 1 *)
    vTestCase1_xp : ARRAY[0..70] OF LWORD;  (* Array data 2 of test case 1 *)
    vTestCase2_act : ARRAY[0..70] OF LWORD;  (* Array data 3 of test case 2 *)
    vTestCase2_xp : ARRAY[0..70] OF LWORD;  (* Array data 4 of test case 2 *)
    i : UINT;  (* Iterator variable i *)
    j : UINT;  (* Iterator variable j *)
  END_VAR

                    (*Run the test cases*)
TEST_CASE_1_SETUP();
TEST_CASE_1_EXEC();

TEST_CASE_2_SETUP();
TEST_CASE_2_EXEC();

(*Instantiate the test runner*)
testRunner(
	Id := 142,
	Name := 'assertArrayEqual_LWORD',
    RunTests := GVL.RunAll OR vRunAll,
	ResetTests := GVL.ResetAll OR vResetAll,
	TestCases:=vTestCases);

(*Report the results to the collection global*)
GVL.Results[testRunner.Id] := testRunner.Summary;
                  

ACTION TEST_CASE_2_SETUP:
                        IF vTestCases[1].state = utTestCaseStates.ut_SETUP THEN
	(*Setup the test case information*)
	vTestCases[1].id := 2;
	vTestCases[1].desc[0] := 'RETURNS FALSE WHEN ARRAYS NOT EQUAL';
    vTestCases[1].desc[1] := 'Tests if the function returns False if the passed in arrays are not identical';
	vTestCases[1].desc[2] := 'PASS IF: Return value is FALSE';
	
	(*Setup needed variables*)
	FOR j:=0 TO 70 DO
		vTestCase2_act[j] := UINT_TO_LWORD(35 * BOOL_TO_UINT(j MOD 2 = 0));
		vTestCase2_xp[j] := UINT_TO_LWORD(35 * BOOL_TO_UINT(j MOD 2 <> 0));
	END_FOR
END_IF
                      
END_ACTION

ACTION TEST_CASE_2_EXEC:
                        IF vTestCases[1].state = utTestCaseStates.ut_RUNNING THEN
	(*Run the test case*)
	IF NOT assertArrayEqual_LWORD(ADR(vTestCase2_act), ADR(vTestCase2_xp), SIZEOF(vTestCase2_act)) THEN
		vTestCases[1].state := utTestCaseStates.ut_PASSED;
		vTestCases[1].msg := 'Arrays were not equal and function returned FALSE -> PASS';
	ELSE
		vTestCases[1].state := utTestCaseStates.ut_FAILED;
		vTestCases[1].msg := 'Arrays were not equal and function returned TRUE -> FAIL';
	END_IF
END_IF
                      
END_ACTION

ACTION TEST_CASE_1_SETUP:
                        IF vTestCases[0].state = utTestCaseStates.ut_SETUP THEN
	(*Setup the test case information*)
	vTestCases[0].id := 1;
	vTestCases[0].desc[0] := 'RETURNS TRUE WHEN ARRAYS EQUAL';
    vTestCases[0].desc[1] := 'Tests if the function returns True if the passed in arrays are identical';
	vTestCases[0].desc[2] := 'PASS IF: Return value is TRUE';
	
	(*Setup needed variables*)
	FOR i:=0 TO 70 DO
		vTestCase1_act[i] := UINT_TO_LWORD(35 * BOOL_TO_UINT(i MOD 2 = 0));
		vTestCase1_xp[i] := UINT_TO_LWORD(35 * BOOL_TO_UINT(i MOD 2 = 0));
	END_FOR
END_IF
                      
END_ACTION

ACTION TEST_CASE_1_EXEC:
                        IF vTestCases[0].state = utTestCaseStates.ut_RUNNING THEN
	(*Run the test case*)
	IF assertArrayEqual_LWORD(ADR(vTestCase1_act), ADR(vTestCase1_xp), SIZEOF(vTestCase1_act)) THEN
		vTestCases[0].state := utTestCaseStates.ut_PASSED;
		vTestCases[0].msg := 'Arrays were equal and function returned TRUE -> PASS';
	ELSE
		vTestCases[0].state := utTestCaseStates.ut_FAILED;
		vTestCases[0].msg := 'Arrays were equal and function returned FALSE -> FAIL';
	END_IF
END_IF
                      
END_ACTION
END_PROGRAM

PROGRAM test_assertLessEqual_TIME_OF_DAY
  VAR
    vTestCases : ARRAY[0..20] OF utTestCase;  (* Definition of all test cases for this POU *)
    testRunner : utTestSuite;  (* Test Suite fb instance to run the tests *)
    vRunAll : BOOL;  (* Manual command to run all tests for this POU *)
    vResetAll : BOOL;  (* Manual command to reset all tests for this POU *)
    vTestCase1_act : TOD;  (* Test data 1 of test case 1 *)
    vTestCase1_xp : TOD;  (* Test data 2 of test case 1 *)
    vTestCase2_act : TOD;  (* Test data 1 of test case 2 *)
    vTestCase2_xp : TOD;  (* Test data 2 of test case 2 *)
    vTestCase3_act : TOD;  (* Test data 1 of test case 3 *)
    vTestCase3_xp : TOD;  (* Test data 2 of test case 3 *)
  END_VAR

                    (*Run the test cases*)
TEST_CASE_1_SETUP();
TEST_CASE_1_EXEC();

TEST_CASE_2_SETUP();
TEST_CASE_2_EXEC();

TEST_CASE_3_SETUP();
TEST_CASE_3_EXEC();

(*Instantiate the test runner*)
testRunner(
	Id := 136,
	Name := 'assertLessEqual_TIME_OF_DAY',
    RunTests := GVL.RunAll OR vRunAll,
	ResetTests := GVL.ResetAll OR vResetAll,
	TestCases:=vTestCases);

(*Report the results to the collection global*)
GVL.Results[testRunner.Id] := testRunner.Summary;
                  

ACTION TEST_CASE_3_SETUP:
                        IF vTestCases[2].state = utTestCaseStates.ut_SETUP THEN
	(*Setup the test case information*)
	vTestCases[2].id := 3;
    vTestCases[2].desc[0] := 'RETURNS FALSE WHEN PARAMETER ACT GREATER THAN XP';
    vTestCases[2].desc[1] := 'Tests if the function returns False if the parameter act is greater than parameter xp';
	vTestCases[2].desc[2] := 'PASS IF: Return value is FALSE';
	
	(*Setup needed variables*)
	vTestCase3_act := REAL_TO_TOD(115.4);
	vTestCase3_xp := REAL_TO_TOD(85.4);
END_IF
                      
END_ACTION

ACTION TEST_CASE_3_EXEC:
                        IF vTestCases[2].state = utTestCaseStates.ut_RUNNING THEN
	(*Run the test case*)
	IF NOT assertLessEqual_TIME_OF_DAY(vTestCase3_act, vTestCase3_xp) THEN
		vTestCases[2].state := utTestCaseStates.ut_PASSED;
		vTestCases[2].msg := 'Parameter act was greater than xp and function returned FALSE -> PASS';
	ELSE
		vTestCases[2].state := utTestCaseStates.ut_FAILED;
		vTestCases[2].msg := 'Parameter act was greater than xp and function returned TRUE -> FAIL';
	END_IF
END_IF
                      
END_ACTION

ACTION TEST_CASE_1_SETUP:
                        IF vTestCases[0].state = utTestCaseStates.ut_SETUP THEN
	(*Setup the test case information*)
	vTestCases[0].id := 1;
	vTestCases[0].desc[0] := 'RETURNS TRUE WHEN PARAMETER ACT LESS THAN XP';
    vTestCases[0].desc[1] := 'Tests if the function returns True if the parameter act is less than parameter xp';
	vTestCases[0].desc[2] := 'PASS IF: Return value is TRUE';
	
	(*Setup needed variables*)
	vTestCase1_act := REAL_TO_TOD(85.4);
	vTestCase1_xp := REAL_TO_TOD(115.4);
END_IF
                      
END_ACTION

ACTION TEST_CASE_1_EXEC:
                        IF vTestCases[0].state = utTestCaseStates.ut_RUNNING THEN
	(*Run the test case*)
	IF assertLessEqual_TIME_OF_DAY(vTestCase1_act, vTestCase1_xp) THEN
		vTestCases[0].state := utTestCaseStates.ut_PASSED;
		vTestCases[0].msg := 'Parameter act was less than xp and function returned TRUE -> PASS';
	ELSE
		vTestCases[0].state := utTestCaseStates.ut_FAILED;
		vTestCases[0].msg := 'Parameter act was less than xp and function returned FALSE -> FAIL';
	END_IF
END_IF
                      
END_ACTION

ACTION TEST_CASE_2_SETUP:
                        IF vTestCases[1].state = utTestCaseStates.ut_SETUP THEN
	(*Setup the test case information*)
	vTestCases[1].id := 2;
    vTestCases[1].desc[0] := 'RETURNS TRUE WHEN PARAMETER ACT EQUAL TO XP';
    vTestCases[1].desc[1] := 'Tests if the function returns True if the parameter act is equal to parameter xp';
	vTestCases[1].desc[2] := 'PASS IF: Return value is TRUE';
	
	(*Setup needed variables*)
	vTestCase2_act := REAL_TO_TOD(115.4);
	vTestCase2_xp := REAL_TO_TOD(115.4);
END_IF
                      
END_ACTION

ACTION TEST_CASE_2_EXEC:
                        IF vTestCases[1].state = utTestCaseStates.ut_RUNNING THEN
	(*Run the test case*)
	IF assertLessEqual_TIME_OF_DAY(vTestCase2_act, vTestCase2_xp) THEN
		vTestCases[1].state := utTestCaseStates.ut_PASSED;
		vTestCases[1].msg := 'Parameter act was equal to xp and function returned TRUE -> PASS';
	ELSE
		vTestCases[1].state := utTestCaseStates.ut_FAILED;
		vTestCases[1].msg := 'Parameter act was equal to xp and function returned FALSE -> FAIL';
	END_IF
END_IF
                      
END_ACTION
END_PROGRAM

PROGRAM test_assertArrayEqual_INT
  VAR
    vTestCases : ARRAY[0..20] OF utTestCase;  (* Definition of all test cases for this POU *)
    testRunner : utTestSuite;  (* Test Suite fb instance to run the tests *)
    vRunAll : BOOL;  (* Manual command to run all tests for this POU *)
    vResetAll : BOOL;  (* Manual command to reset all tests for this POU *)
    vTestCase1_act : ARRAY[0..70] OF INT;  (* Array data 1 of test case 1 *)
    vTestCase1_xp : ARRAY[0..70] OF INT;  (* Array data 2 of test case 1 *)
    vTestCase2_act : ARRAY[0..70] OF INT;  (* Array data 3 of test case 2 *)
    vTestCase2_xp : ARRAY[0..70] OF INT;  (* Array data 4 of test case 2 *)
    i : UINT;  (* Iterator variable i *)
    j : UINT;  (* Iterator variable j *)
  END_VAR

                    (*Run the test cases*)
TEST_CASE_1_SETUP();
TEST_CASE_1_EXEC();

TEST_CASE_2_SETUP();
TEST_CASE_2_EXEC();

(*Instantiate the test runner*)
testRunner(
	Id := 145,
	Name := 'assertArrayEqual_INT',
    RunTests := GVL.RunAll OR vRunAll,
	ResetTests := GVL.ResetAll OR vResetAll,
	TestCases:=vTestCases);

(*Report the results to the collection global*)
GVL.Results[testRunner.Id] := testRunner.Summary;
                  

ACTION TEST_CASE_1_EXEC:
                        IF vTestCases[0].state = utTestCaseStates.ut_RUNNING THEN
	(*Run the test case*)
	IF assertArrayEqual_INT(ADR(vTestCase1_act), ADR(vTestCase1_xp), SIZEOF(vTestCase1_act)) THEN
		vTestCases[0].state := utTestCaseStates.ut_PASSED;
		vTestCases[0].msg := 'Arrays were equal and function returned TRUE -> PASS';
	ELSE
		vTestCases[0].state := utTestCaseStates.ut_FAILED;
		vTestCases[0].msg := 'Arrays were equal and function returned FALSE -> FAIL';
	END_IF
END_IF
                      
END_ACTION

ACTION TEST_CASE_1_SETUP:
                        IF vTestCases[0].state = utTestCaseStates.ut_SETUP THEN
	(*Setup the test case information*)
	vTestCases[0].id := 1;
	vTestCases[0].desc[0] := 'RETURNS TRUE WHEN ARRAYS EQUAL';
    vTestCases[0].desc[1] := 'Tests if the function returns True if the passed in arrays are identical';
	vTestCases[0].desc[2] := 'PASS IF: Return value is TRUE';
	
	(*Setup needed variables*)
	FOR i:=0 TO 70 DO
		vTestCase1_act[i] := UINT_TO_INT(35 * BOOL_TO_UINT(i MOD 2 = 0));
		vTestCase1_xp[i] := UINT_TO_INT(35 * BOOL_TO_UINT(i MOD 2 = 0));
	END_FOR
END_IF
                      
END_ACTION

ACTION TEST_CASE_2_SETUP:
                        IF vTestCases[1].state = utTestCaseStates.ut_SETUP THEN
	(*Setup the test case information*)
	vTestCases[1].id := 2;
	vTestCases[1].desc[0] := 'RETURNS FALSE WHEN ARRAYS NOT EQUAL';
    vTestCases[1].desc[1] := 'Tests if the function returns False if the passed in arrays are not identical';
	vTestCases[1].desc[2] := 'PASS IF: Return value is FALSE';
	
	(*Setup needed variables*)
	FOR j:=0 TO 70 DO
		vTestCase2_act[j] := UINT_TO_INT(35 * BOOL_TO_UINT(j MOD 2 = 0));
		vTestCase2_xp[j] := UINT_TO_INT(35 * BOOL_TO_UINT(j MOD 2 <> 0));
	END_FOR
END_IF
                      
END_ACTION

ACTION TEST_CASE_2_EXEC:
                        IF vTestCases[1].state = utTestCaseStates.ut_RUNNING THEN
	(*Run the test case*)
	IF NOT assertArrayEqual_INT(ADR(vTestCase2_act), ADR(vTestCase2_xp), SIZEOF(vTestCase2_act)) THEN
		vTestCases[1].state := utTestCaseStates.ut_PASSED;
		vTestCases[1].msg := 'Arrays were not equal and function returned FALSE -> PASS';
	ELSE
		vTestCases[1].state := utTestCaseStates.ut_FAILED;
		vTestCases[1].msg := 'Arrays were not equal and function returned TRUE -> FAIL';
	END_IF
END_IF
                      
END_ACTION
END_PROGRAM

PROGRAM test_assertArrayEqual_BOOL
  VAR
    vTestCases : ARRAY[0..20] OF utTestCase;  (* Definition of all test cases for this POU *)
    testRunner : utTestSuite;  (* Test Suite fb instance to run the tests *)
    vRunAll : BOOL;  (* Manual command to run all tests for this POU *)
    vResetAll : BOOL;  (* Manual command to reset all tests for this POU *)
    vTestCase1_act : ARRAY[0..70] OF BOOL;  (* Array data 1 of test case 1 *)
    vTestCase1_xp : ARRAY[0..70] OF BOOL;  (* Array data 2 of test case 1 *)
    vTestCase2_act : ARRAY[0..70] OF BOOL;  (* Array data 3 of test case 2 *)
    vTestCase2_xp : ARRAY[0..70] OF BOOL;  (* Array data 4 of test case 2 *)
    i : UINT;  (* Iterator variable i *)
    j : UINT;  (* Iterator variable j *)
  END_VAR

                    (*Run the test cases*)
TEST_CASE_1_SETUP();
TEST_CASE_1_EXEC();

TEST_CASE_2_SETUP();
TEST_CASE_2_EXEC();

(*Instantiate the test runner*)
testRunner(
	Id := 138,
	Name := 'assertArrayEqual_BOOL',
    RunTests := GVL.RunAll OR vRunAll,
	ResetTests := GVL.ResetAll OR vResetAll,
	TestCases:=vTestCases);

(*Report the results to the collection global*)
GVL.Results[testRunner.Id] := testRunner.Summary;
                  

ACTION TEST_CASE_1_EXEC:
                        IF vTestCases[0].state = utTestCaseStates.ut_RUNNING THEN
	(*Run the test case*)
	IF assertArrayEqual_BOOL(ADR(vTestCase1_act), ADR(vTestCase1_xp), SIZEOF(vTestCase1_act)) THEN
		vTestCases[0].state := utTestCaseStates.ut_PASSED;
		vTestCases[0].msg := 'Arrays were equal and function returned TRUE -> PASS';
	ELSE
		vTestCases[0].state := utTestCaseStates.ut_FAILED;
		vTestCases[0].msg := 'Arrays were equal and function returned FALSE -> FAIL';
	END_IF
END_IF
                      
END_ACTION

ACTION TEST_CASE_1_SETUP:
                        IF vTestCases[0].state = utTestCaseStates.ut_SETUP THEN
	(*Setup the test case information*)
	vTestCases[0].id := 1;
	vTestCases[0].desc[0] := 'RETURNS TRUE WHEN ARRAYS EQUAL';
    vTestCases[0].desc[1] := 'Tests if the function returns True if the passed in arrays are identical';
	vTestCases[0].desc[2] := 'PASS IF: Return value is TRUE';
	
	(*Setup needed variables*)
	FOR i:=0 TO 70 DO
		vTestCase1_act[i] := UINT_TO_BOOL(35 * BOOL_TO_UINT(i MOD 2 = 0));
		vTestCase1_xp[i] := UINT_TO_BOOL(35 * BOOL_TO_UINT(i MOD 2 = 0));
	END_FOR
END_IF
                      
END_ACTION

ACTION TEST_CASE_2_SETUP:
                        IF vTestCases[1].state = utTestCaseStates.ut_SETUP THEN
	(*Setup the test case information*)
	vTestCases[1].id := 2;
	vTestCases[1].desc[0] := 'RETURNS FALSE WHEN ARRAYS NOT EQUAL';
    vTestCases[1].desc[1] := 'Tests if the function returns False if the passed in arrays are not identical';
	vTestCases[1].desc[2] := 'PASS IF: Return value is FALSE';
	
	(*Setup needed variables*)
	FOR j:=0 TO 70 DO
		vTestCase2_act[j] := UINT_TO_BOOL(35 * BOOL_TO_UINT(j MOD 2 = 0));
		vTestCase2_xp[j] := UINT_TO_BOOL(35 * BOOL_TO_UINT(j MOD 2 <> 0));
	END_FOR
END_IF
                      
END_ACTION

ACTION TEST_CASE_2_EXEC:
                        IF vTestCases[1].state = utTestCaseStates.ut_RUNNING THEN
	(*Run the test case*)
	IF NOT assertArrayEqual_BOOL(ADR(vTestCase2_act), ADR(vTestCase2_xp), SIZEOF(vTestCase2_act)) THEN
		vTestCases[1].state := utTestCaseStates.ut_PASSED;
		vTestCases[1].msg := 'Arrays were not equal and function returned FALSE -> PASS';
	ELSE
		vTestCases[1].state := utTestCaseStates.ut_FAILED;
		vTestCases[1].msg := 'Arrays were not equal and function returned TRUE -> FAIL';
	END_IF
END_IF
                      
END_ACTION
END_PROGRAM

PROGRAM test_assertLessEqual_UDINT
  VAR
    vTestCases : ARRAY[0..20] OF utTestCase;  (* Definition of all test cases for this POU *)
    testRunner : utTestSuite;  (* Test Suite fb instance to run the tests *)
    vRunAll : BOOL;  (* Manual command to run all tests for this POU *)
    vResetAll : BOOL;  (* Manual command to reset all tests for this POU *)
    vTestCase1_act : UDINT;  (* Test data 1 of test case 1 *)
    vTestCase1_xp : UDINT;  (* Test data 2 of test case 1 *)
    vTestCase2_act : UDINT;  (* Test data 1 of test case 2 *)
    vTestCase2_xp : UDINT;  (* Test data 2 of test case 2 *)
    vTestCase3_act : UDINT;  (* Test data 1 of test case 3 *)
    vTestCase3_xp : UDINT;  (* Test data 2 of test case 3 *)
  END_VAR

                    (*Run the test cases*)
TEST_CASE_1_SETUP();
TEST_CASE_1_EXEC();

TEST_CASE_2_SETUP();
TEST_CASE_2_EXEC();

TEST_CASE_3_SETUP();
TEST_CASE_3_EXEC();

(*Instantiate the test runner*)
testRunner(
	Id := 125,
	Name := 'assertLessEqual_UDINT',
    RunTests := GVL.RunAll OR vRunAll,
	ResetTests := GVL.ResetAll OR vResetAll,
	TestCases:=vTestCases);

(*Report the results to the collection global*)
GVL.Results[testRunner.Id] := testRunner.Summary;
                  

ACTION TEST_CASE_3_EXEC:
                        IF vTestCases[2].state = utTestCaseStates.ut_RUNNING THEN
	(*Run the test case*)
	IF NOT assertLessEqual_UDINT(vTestCase3_act, vTestCase3_xp) THEN
		vTestCases[2].state := utTestCaseStates.ut_PASSED;
		vTestCases[2].msg := 'Parameter act was greater than xp and function returned FALSE -> PASS';
	ELSE
		vTestCases[2].state := utTestCaseStates.ut_FAILED;
		vTestCases[2].msg := 'Parameter act was greater than xp and function returned TRUE -> FAIL';
	END_IF
END_IF
                      
END_ACTION

ACTION TEST_CASE_2_EXEC:
                        IF vTestCases[1].state = utTestCaseStates.ut_RUNNING THEN
	(*Run the test case*)
	IF assertLessEqual_UDINT(vTestCase2_act, vTestCase2_xp) THEN
		vTestCases[1].state := utTestCaseStates.ut_PASSED;
		vTestCases[1].msg := 'Parameter act was equal to xp and function returned TRUE -> PASS';
	ELSE
		vTestCases[1].state := utTestCaseStates.ut_FAILED;
		vTestCases[1].msg := 'Parameter act was equal to xp and function returned FALSE -> FAIL';
	END_IF
END_IF
                      
END_ACTION

ACTION TEST_CASE_3_SETUP:
                        IF vTestCases[2].state = utTestCaseStates.ut_SETUP THEN
	(*Setup the test case information*)
	vTestCases[2].id := 3;
    vTestCases[2].desc[0] := 'RETURNS FALSE WHEN PARAMETER ACT GREATER THAN XP';
    vTestCases[2].desc[1] := 'Tests if the function returns False if the parameter act is greater than parameter xp';
	vTestCases[2].desc[2] := 'PASS IF: Return value is FALSE';
	
	(*Setup needed variables*)
	vTestCase3_act := REAL_TO_UDINT(115.4);
	vTestCase3_xp := REAL_TO_UDINT(85.4);
END_IF
                      
END_ACTION

ACTION TEST_CASE_1_SETUP:
                        IF vTestCases[0].state = utTestCaseStates.ut_SETUP THEN
	(*Setup the test case information*)
	vTestCases[0].id := 1;
	vTestCases[0].desc[0] := 'RETURNS TRUE WHEN PARAMETER ACT LESS THAN XP';
    vTestCases[0].desc[1] := 'Tests if the function returns True if the parameter act is less than parameter xp';
	vTestCases[0].desc[2] := 'PASS IF: Return value is TRUE';
	
	(*Setup needed variables*)
	vTestCase1_act := REAL_TO_UDINT(85.4);
	vTestCase1_xp := REAL_TO_UDINT(115.4);
END_IF
                      
END_ACTION

ACTION TEST_CASE_1_EXEC:
                        IF vTestCases[0].state = utTestCaseStates.ut_RUNNING THEN
	(*Run the test case*)
	IF assertLessEqual_UDINT(vTestCase1_act, vTestCase1_xp) THEN
		vTestCases[0].state := utTestCaseStates.ut_PASSED;
		vTestCases[0].msg := 'Parameter act was less than xp and function returned TRUE -> PASS';
	ELSE
		vTestCases[0].state := utTestCaseStates.ut_FAILED;
		vTestCases[0].msg := 'Parameter act was less than xp and function returned FALSE -> FAIL';
	END_IF
END_IF
                      
END_ACTION

ACTION TEST_CASE_2_SETUP:
                        IF vTestCases[1].state = utTestCaseStates.ut_SETUP THEN
	(*Setup the test case information*)
	vTestCases[1].id := 2;
    vTestCases[1].desc[0] := 'RETURNS TRUE WHEN PARAMETER ACT EQUAL TO XP';
    vTestCases[1].desc[1] := 'Tests if the function returns True if the parameter act is equal to parameter xp';
	vTestCases[1].desc[2] := 'PASS IF: Return value is TRUE';
	
	(*Setup needed variables*)
	vTestCase2_act := REAL_TO_UDINT(115.4);
	vTestCase2_xp := REAL_TO_UDINT(115.4);
END_IF
                      
END_ACTION
END_PROGRAM

PROGRAM test_assertLessEqual_DATE
  VAR
    vTestCases : ARRAY[0..20] OF utTestCase;  (* Definition of all test cases for this POU *)
    testRunner : utTestSuite;  (* Test Suite fb instance to run the tests *)
    vRunAll : BOOL;  (* Manual command to run all tests for this POU *)
    vResetAll : BOOL;  (* Manual command to reset all tests for this POU *)
    vTestCase1_act : DATE;  (* Test data 1 of test case 1 *)
    vTestCase1_xp : DATE;  (* Test data 2 of test case 1 *)
    vTestCase2_act : DATE;  (* Test data 1 of test case 2 *)
    vTestCase2_xp : DATE;  (* Test data 2 of test case 2 *)
    vTestCase3_act : DATE;  (* Test data 1 of test case 3 *)
    vTestCase3_xp : DATE;  (* Test data 2 of test case 3 *)
  END_VAR

                    (*Run the test cases*)
TEST_CASE_1_SETUP();
TEST_CASE_1_EXEC();

TEST_CASE_2_SETUP();
TEST_CASE_2_EXEC();

TEST_CASE_3_SETUP();
TEST_CASE_3_EXEC();

(*Instantiate the test runner*)
testRunner(
	Id := 132,
	Name := 'assertLessEqual_DATE',
    RunTests := GVL.RunAll OR vRunAll,
	ResetTests := GVL.ResetAll OR vResetAll,
	TestCases:=vTestCases);

(*Report the results to the collection global*)
GVL.Results[testRunner.Id] := testRunner.Summary;
                  

ACTION TEST_CASE_3_EXEC:
                        IF vTestCases[2].state = utTestCaseStates.ut_RUNNING THEN
	(*Run the test case*)
	IF NOT assertLessEqual_DATE(vTestCase3_act, vTestCase3_xp) THEN
		vTestCases[2].state := utTestCaseStates.ut_PASSED;
		vTestCases[2].msg := 'Parameter act was greater than xp and function returned FALSE -> PASS';
	ELSE
		vTestCases[2].state := utTestCaseStates.ut_FAILED;
		vTestCases[2].msg := 'Parameter act was greater than xp and function returned TRUE -> FAIL';
	END_IF
END_IF
                      
END_ACTION

ACTION TEST_CASE_2_EXEC:
                        IF vTestCases[1].state = utTestCaseStates.ut_RUNNING THEN
	(*Run the test case*)
	IF assertLessEqual_DATE(vTestCase2_act, vTestCase2_xp) THEN
		vTestCases[1].state := utTestCaseStates.ut_PASSED;
		vTestCases[1].msg := 'Parameter act was equal to xp and function returned TRUE -> PASS';
	ELSE
		vTestCases[1].state := utTestCaseStates.ut_FAILED;
		vTestCases[1].msg := 'Parameter act was equal to xp and function returned FALSE -> FAIL';
	END_IF
END_IF
                      
END_ACTION

ACTION TEST_CASE_3_SETUP:
                        IF vTestCases[2].state = utTestCaseStates.ut_SETUP THEN
	(*Setup the test case information*)
	vTestCases[2].id := 3;
    vTestCases[2].desc[0] := 'RETURNS FALSE WHEN PARAMETER ACT GREATER THAN XP';
    vTestCases[2].desc[1] := 'Tests if the function returns False if the parameter act is greater than parameter xp';
	vTestCases[2].desc[2] := 'PASS IF: Return value is FALSE';
	
	(*Setup needed variables*)
	vTestCase3_act := REAL_TO_DATE(115.4);
	vTestCase3_xp := REAL_TO_DATE(85.4);
END_IF
                      
END_ACTION

ACTION TEST_CASE_1_SETUP:
                        IF vTestCases[0].state = utTestCaseStates.ut_SETUP THEN
	(*Setup the test case information*)
	vTestCases[0].id := 1;
	vTestCases[0].desc[0] := 'RETURNS TRUE WHEN PARAMETER ACT LESS THAN XP';
    vTestCases[0].desc[1] := 'Tests if the function returns True if the parameter act is less than parameter xp';
	vTestCases[0].desc[2] := 'PASS IF: Return value is TRUE';
	
	(*Setup needed variables*)
	vTestCase1_act := REAL_TO_DATE(85.4);
	vTestCase1_xp := REAL_TO_DATE(115.4);
END_IF
                      
END_ACTION

ACTION TEST_CASE_1_EXEC:
                        IF vTestCases[0].state = utTestCaseStates.ut_RUNNING THEN
	(*Run the test case*)
	IF assertLessEqual_DATE(vTestCase1_act, vTestCase1_xp) THEN
		vTestCases[0].state := utTestCaseStates.ut_PASSED;
		vTestCases[0].msg := 'Parameter act was less than xp and function returned TRUE -> PASS';
	ELSE
		vTestCases[0].state := utTestCaseStates.ut_FAILED;
		vTestCases[0].msg := 'Parameter act was less than xp and function returned FALSE -> FAIL';
	END_IF
END_IF
                      
END_ACTION

ACTION TEST_CASE_2_SETUP:
                        IF vTestCases[1].state = utTestCaseStates.ut_SETUP THEN
	(*Setup the test case information*)
	vTestCases[1].id := 2;
    vTestCases[1].desc[0] := 'RETURNS TRUE WHEN PARAMETER ACT EQUAL TO XP';
    vTestCases[1].desc[1] := 'Tests if the function returns True if the parameter act is equal to parameter xp';
	vTestCases[1].desc[2] := 'PASS IF: Return value is TRUE';
	
	(*Setup needed variables*)
	vTestCase2_act := REAL_TO_DATE(115.4);
	vTestCase2_xp := REAL_TO_DATE(115.4);
END_IF
                      
END_ACTION
END_PROGRAM

PROGRAM test_assertLessEqual_LINT
  VAR
    vTestCases : ARRAY[0..20] OF utTestCase;  (* Definition of all test cases for this POU *)
    testRunner : utTestSuite;  (* Test Suite fb instance to run the tests *)
    vRunAll : BOOL;  (* Manual command to run all tests for this POU *)
    vResetAll : BOOL;  (* Manual command to reset all tests for this POU *)
    vTestCase1_act : LINT;  (* Test data 1 of test case 1 *)
    vTestCase1_xp : LINT;  (* Test data 2 of test case 1 *)
    vTestCase2_act : LINT;  (* Test data 1 of test case 2 *)
    vTestCase2_xp : LINT;  (* Test data 2 of test case 2 *)
    vTestCase3_act : LINT;  (* Test data 1 of test case 3 *)
    vTestCase3_xp : LINT;  (* Test data 2 of test case 3 *)
  END_VAR

                    (*Run the test cases*)
TEST_CASE_1_SETUP();
TEST_CASE_1_EXEC();

TEST_CASE_2_SETUP();
TEST_CASE_2_EXEC();

TEST_CASE_3_SETUP();
TEST_CASE_3_EXEC();

(*Instantiate the test runner*)
testRunner(
	Id := 126,
	Name := 'assertLessEqual_LINT',
    RunTests := GVL.RunAll OR vRunAll,
	ResetTests := GVL.ResetAll OR vResetAll,
	TestCases:=vTestCases);

(*Report the results to the collection global*)
GVL.Results[testRunner.Id] := testRunner.Summary;
                  

ACTION TEST_CASE_3_SETUP:
                        IF vTestCases[2].state = utTestCaseStates.ut_SETUP THEN
	(*Setup the test case information*)
	vTestCases[2].id := 3;
    vTestCases[2].desc[0] := 'RETURNS FALSE WHEN PARAMETER ACT GREATER THAN XP';
    vTestCases[2].desc[1] := 'Tests if the function returns False if the parameter act is greater than parameter xp';
	vTestCases[2].desc[2] := 'PASS IF: Return value is FALSE';
	
	(*Setup needed variables*)
	vTestCase3_act := REAL_TO_LINT(115.4);
	vTestCase3_xp := REAL_TO_LINT(85.4);
END_IF
                      
END_ACTION

ACTION TEST_CASE_3_EXEC:
                        IF vTestCases[2].state = utTestCaseStates.ut_RUNNING THEN
	(*Run the test case*)
	IF NOT assertLessEqual_LINT(vTestCase3_act, vTestCase3_xp) THEN
		vTestCases[2].state := utTestCaseStates.ut_PASSED;
		vTestCases[2].msg := 'Parameter act was greater than xp and function returned FALSE -> PASS';
	ELSE
		vTestCases[2].state := utTestCaseStates.ut_FAILED;
		vTestCases[2].msg := 'Parameter act was greater than xp and function returned TRUE -> FAIL';
	END_IF
END_IF
                      
END_ACTION

ACTION TEST_CASE_1_SETUP:
                        IF vTestCases[0].state = utTestCaseStates.ut_SETUP THEN
	(*Setup the test case information*)
	vTestCases[0].id := 1;
	vTestCases[0].desc[0] := 'RETURNS TRUE WHEN PARAMETER ACT LESS THAN XP';
    vTestCases[0].desc[1] := 'Tests if the function returns True if the parameter act is less than parameter xp';
	vTestCases[0].desc[2] := 'PASS IF: Return value is TRUE';
	
	(*Setup needed variables*)
	vTestCase1_act := REAL_TO_LINT(85.4);
	vTestCase1_xp := REAL_TO_LINT(115.4);
END_IF
                      
END_ACTION

ACTION TEST_CASE_1_EXEC:
                        IF vTestCases[0].state = utTestCaseStates.ut_RUNNING THEN
	(*Run the test case*)
	IF assertLessEqual_LINT(vTestCase1_act, vTestCase1_xp) THEN
		vTestCases[0].state := utTestCaseStates.ut_PASSED;
		vTestCases[0].msg := 'Parameter act was less than xp and function returned TRUE -> PASS';
	ELSE
		vTestCases[0].state := utTestCaseStates.ut_FAILED;
		vTestCases[0].msg := 'Parameter act was less than xp and function returned FALSE -> FAIL';
	END_IF
END_IF
                      
END_ACTION

ACTION TEST_CASE_2_SETUP:
                        IF vTestCases[1].state = utTestCaseStates.ut_SETUP THEN
	(*Setup the test case information*)
	vTestCases[1].id := 2;
    vTestCases[1].desc[0] := 'RETURNS TRUE WHEN PARAMETER ACT EQUAL TO XP';
    vTestCases[1].desc[1] := 'Tests if the function returns True if the parameter act is equal to parameter xp';
	vTestCases[1].desc[2] := 'PASS IF: Return value is TRUE';
	
	(*Setup needed variables*)
	vTestCase2_act := REAL_TO_LINT(115.4);
	vTestCase2_xp := REAL_TO_LINT(115.4);
END_IF
                      
END_ACTION

ACTION TEST_CASE_2_EXEC:
                        IF vTestCases[1].state = utTestCaseStates.ut_RUNNING THEN
	(*Run the test case*)
	IF assertLessEqual_LINT(vTestCase2_act, vTestCase2_xp) THEN
		vTestCases[1].state := utTestCaseStates.ut_PASSED;
		vTestCases[1].msg := 'Parameter act was equal to xp and function returned TRUE -> PASS';
	ELSE
		vTestCases[1].state := utTestCaseStates.ut_FAILED;
		vTestCases[1].msg := 'Parameter act was equal to xp and function returned FALSE -> FAIL';
	END_IF
END_IF
                      
END_ACTION
END_PROGRAM

PROGRAM test_assertLessEqual_ULINT
  VAR
    vTestCases : ARRAY[0..20] OF utTestCase;  (* Definition of all test cases for this POU *)
    testRunner : utTestSuite;  (* Test Suite fb instance to run the tests *)
    vRunAll : BOOL;  (* Manual command to run all tests for this POU *)
    vResetAll : BOOL;  (* Manual command to reset all tests for this POU *)
    vTestCase1_act : ULINT;  (* Test data 1 of test case 1 *)
    vTestCase1_xp : ULINT;  (* Test data 2 of test case 1 *)
    vTestCase2_act : ULINT;  (* Test data 1 of test case 2 *)
    vTestCase2_xp : ULINT;  (* Test data 2 of test case 2 *)
    vTestCase3_act : ULINT;  (* Test data 1 of test case 3 *)
    vTestCase3_xp : ULINT;  (* Test data 2 of test case 3 *)
  END_VAR

                    (*Run the test cases*)
TEST_CASE_1_SETUP();
TEST_CASE_1_EXEC();

TEST_CASE_2_SETUP();
TEST_CASE_2_EXEC();

TEST_CASE_3_SETUP();
TEST_CASE_3_EXEC();

(*Instantiate the test runner*)
testRunner(
	Id := 127,
	Name := 'assertLessEqual_ULINT',
    RunTests := GVL.RunAll OR vRunAll,
	ResetTests := GVL.ResetAll OR vResetAll,
	TestCases:=vTestCases);

(*Report the results to the collection global*)
GVL.Results[testRunner.Id] := testRunner.Summary;
                  

ACTION TEST_CASE_1_SETUP:
                        IF vTestCases[0].state = utTestCaseStates.ut_SETUP THEN
	(*Setup the test case information*)
	vTestCases[0].id := 1;
	vTestCases[0].desc[0] := 'RETURNS TRUE WHEN PARAMETER ACT LESS THAN XP';
    vTestCases[0].desc[1] := 'Tests if the function returns True if the parameter act is less than parameter xp';
	vTestCases[0].desc[2] := 'PASS IF: Return value is TRUE';
	
	(*Setup needed variables*)
	vTestCase1_act := REAL_TO_ULINT(85.4);
	vTestCase1_xp := REAL_TO_ULINT(115.4);
END_IF
                      
END_ACTION

ACTION TEST_CASE_3_SETUP:
                        IF vTestCases[2].state = utTestCaseStates.ut_SETUP THEN
	(*Setup the test case information*)
	vTestCases[2].id := 3;
    vTestCases[2].desc[0] := 'RETURNS FALSE WHEN PARAMETER ACT GREATER THAN XP';
    vTestCases[2].desc[1] := 'Tests if the function returns False if the parameter act is greater than parameter xp';
	vTestCases[2].desc[2] := 'PASS IF: Return value is FALSE';
	
	(*Setup needed variables*)
	vTestCase3_act := REAL_TO_ULINT(115.4);
	vTestCase3_xp := REAL_TO_ULINT(85.4);
END_IF
                      
END_ACTION

ACTION TEST_CASE_3_EXEC:
                        IF vTestCases[2].state = utTestCaseStates.ut_RUNNING THEN
	(*Run the test case*)
	IF NOT assertLessEqual_ULINT(vTestCase3_act, vTestCase3_xp) THEN
		vTestCases[2].state := utTestCaseStates.ut_PASSED;
		vTestCases[2].msg := 'Parameter act was greater than xp and function returned FALSE -> PASS';
	ELSE
		vTestCases[2].state := utTestCaseStates.ut_FAILED;
		vTestCases[2].msg := 'Parameter act was greater than xp and function returned TRUE -> FAIL';
	END_IF
END_IF
                      
END_ACTION

ACTION TEST_CASE_1_EXEC:
                        IF vTestCases[0].state = utTestCaseStates.ut_RUNNING THEN
	(*Run the test case*)
	IF assertLessEqual_ULINT(vTestCase1_act, vTestCase1_xp) THEN
		vTestCases[0].state := utTestCaseStates.ut_PASSED;
		vTestCases[0].msg := 'Parameter act was less than xp and function returned TRUE -> PASS';
	ELSE
		vTestCases[0].state := utTestCaseStates.ut_FAILED;
		vTestCases[0].msg := 'Parameter act was less than xp and function returned FALSE -> FAIL';
	END_IF
END_IF
                      
END_ACTION

ACTION TEST_CASE_2_SETUP:
                        IF vTestCases[1].state = utTestCaseStates.ut_SETUP THEN
	(*Setup the test case information*)
	vTestCases[1].id := 2;
    vTestCases[1].desc[0] := 'RETURNS TRUE WHEN PARAMETER ACT EQUAL TO XP';
    vTestCases[1].desc[1] := 'Tests if the function returns True if the parameter act is equal to parameter xp';
	vTestCases[1].desc[2] := 'PASS IF: Return value is TRUE';
	
	(*Setup needed variables*)
	vTestCase2_act := REAL_TO_ULINT(115.4);
	vTestCase2_xp := REAL_TO_ULINT(115.4);
END_IF
                      
END_ACTION

ACTION TEST_CASE_2_EXEC:
                        IF vTestCases[1].state = utTestCaseStates.ut_RUNNING THEN
	(*Run the test case*)
	IF assertLessEqual_ULINT(vTestCase2_act, vTestCase2_xp) THEN
		vTestCases[1].state := utTestCaseStates.ut_PASSED;
		vTestCases[1].msg := 'Parameter act was equal to xp and function returned TRUE -> PASS';
	ELSE
		vTestCases[1].state := utTestCaseStates.ut_FAILED;
		vTestCases[1].msg := 'Parameter act was equal to xp and function returned FALSE -> FAIL';
	END_IF
END_IF
                      
END_ACTION
END_PROGRAM

PROGRAM test_assertLessEqual_LDATE
  VAR
    vTestCases : ARRAY[0..20] OF utTestCase;  (* Definition of all test cases for this POU *)
    testRunner : utTestSuite;  (* Test Suite fb instance to run the tests *)
    vRunAll : BOOL;  (* Manual command to run all tests for this POU *)
    vResetAll : BOOL;  (* Manual command to reset all tests for this POU *)
    vTestCase1_act : LDATE;  (* Test data 1 of test case 1 *)
    vTestCase1_xp : LDATE;  (* Test data 2 of test case 1 *)
    vTestCase2_act : LDATE;  (* Test data 1 of test case 2 *)
    vTestCase2_xp : LDATE;  (* Test data 2 of test case 2 *)
    vTestCase3_act : LDATE;  (* Test data 1 of test case 3 *)
    vTestCase3_xp : LDATE;  (* Test data 2 of test case 3 *)
  END_VAR

                    (*Run the test cases*)
TEST_CASE_1_SETUP();
TEST_CASE_1_EXEC();

TEST_CASE_2_SETUP();
TEST_CASE_2_EXEC();

TEST_CASE_3_SETUP();
TEST_CASE_3_EXEC();

(*Instantiate the test runner*)
testRunner(
	Id := 133,
	Name := 'assertLessEqual_LDATE',
    RunTests := GVL.RunAll OR vRunAll,
	ResetTests := GVL.ResetAll OR vResetAll,
	TestCases:=vTestCases);

(*Report the results to the collection global*)
GVL.Results[testRunner.Id] := testRunner.Summary;
                  

ACTION TEST_CASE_3_SETUP:
                        IF vTestCases[2].state = utTestCaseStates.ut_SETUP THEN
	(*Setup the test case information*)
	vTestCases[2].id := 3;
    vTestCases[2].desc[0] := 'RETURNS FALSE WHEN PARAMETER ACT GREATER THAN XP';
    vTestCases[2].desc[1] := 'Tests if the function returns False if the parameter act is greater than parameter xp';
	vTestCases[2].desc[2] := 'PASS IF: Return value is FALSE';
	
	(*Setup needed variables*)
	vTestCase3_act := REAL_TO_LDATE(115.4);
	vTestCase3_xp := REAL_TO_LDATE(85.4);
END_IF
                      
END_ACTION

ACTION TEST_CASE_3_EXEC:
                        IF vTestCases[2].state = utTestCaseStates.ut_RUNNING THEN
	(*Run the test case*)
	IF NOT assertLessEqual_LDATE(vTestCase3_act, vTestCase3_xp) THEN
		vTestCases[2].state := utTestCaseStates.ut_PASSED;
		vTestCases[2].msg := 'Parameter act was greater than xp and function returned FALSE -> PASS';
	ELSE
		vTestCases[2].state := utTestCaseStates.ut_FAILED;
		vTestCases[2].msg := 'Parameter act was greater than xp and function returned TRUE -> FAIL';
	END_IF
END_IF
                      
END_ACTION

ACTION TEST_CASE_1_SETUP:
                        IF vTestCases[0].state = utTestCaseStates.ut_SETUP THEN
	(*Setup the test case information*)
	vTestCases[0].id := 1;
	vTestCases[0].desc[0] := 'RETURNS TRUE WHEN PARAMETER ACT LESS THAN XP';
    vTestCases[0].desc[1] := 'Tests if the function returns True if the parameter act is less than parameter xp';
	vTestCases[0].desc[2] := 'PASS IF: Return value is TRUE';
	
	(*Setup needed variables*)
	vTestCase1_act := REAL_TO_LDATE(85.4);
	vTestCase1_xp := REAL_TO_LDATE(115.4);
END_IF
                      
END_ACTION

ACTION TEST_CASE_1_EXEC:
                        IF vTestCases[0].state = utTestCaseStates.ut_RUNNING THEN
	(*Run the test case*)
	IF assertLessEqual_LDATE(vTestCase1_act, vTestCase1_xp) THEN
		vTestCases[0].state := utTestCaseStates.ut_PASSED;
		vTestCases[0].msg := 'Parameter act was less than xp and function returned TRUE -> PASS';
	ELSE
		vTestCases[0].state := utTestCaseStates.ut_FAILED;
		vTestCases[0].msg := 'Parameter act was less than xp and function returned FALSE -> FAIL';
	END_IF
END_IF
                      
END_ACTION

ACTION TEST_CASE_2_SETUP:
                        IF vTestCases[1].state = utTestCaseStates.ut_SETUP THEN
	(*Setup the test case information*)
	vTestCases[1].id := 2;
    vTestCases[1].desc[0] := 'RETURNS TRUE WHEN PARAMETER ACT EQUAL TO XP';
    vTestCases[1].desc[1] := 'Tests if the function returns True if the parameter act is equal to parameter xp';
	vTestCases[1].desc[2] := 'PASS IF: Return value is TRUE';
	
	(*Setup needed variables*)
	vTestCase2_act := REAL_TO_LDATE(115.4);
	vTestCase2_xp := REAL_TO_LDATE(115.4);
END_IF
                      
END_ACTION

ACTION TEST_CASE_2_EXEC:
                        IF vTestCases[1].state = utTestCaseStates.ut_RUNNING THEN
	(*Run the test case*)
	IF assertLessEqual_LDATE(vTestCase2_act, vTestCase2_xp) THEN
		vTestCases[1].state := utTestCaseStates.ut_PASSED;
		vTestCases[1].msg := 'Parameter act was equal to xp and function returned TRUE -> PASS';
	ELSE
		vTestCases[1].state := utTestCaseStates.ut_FAILED;
		vTestCases[1].msg := 'Parameter act was equal to xp and function returned FALSE -> FAIL';
	END_IF
END_IF
                      
END_ACTION
END_PROGRAM

PROGRAM test_assertLessEqual_DATE_AND_TIME
  VAR
    vTestCases : ARRAY[0..20] OF utTestCase;  (* Definition of all test cases for this POU *)
    testRunner : utTestSuite;  (* Test Suite fb instance to run the tests *)
    vRunAll : BOOL;  (* Manual command to run all tests for this POU *)
    vResetAll : BOOL;  (* Manual command to reset all tests for this POU *)
    vTestCase1_act : DT;  (* Test data 1 of test case 1 *)
    vTestCase1_xp : DT;  (* Test data 2 of test case 1 *)
    vTestCase2_act : DT;  (* Test data 1 of test case 2 *)
    vTestCase2_xp : DT;  (* Test data 2 of test case 2 *)
    vTestCase3_act : DT;  (* Test data 1 of test case 3 *)
    vTestCase3_xp : DT;  (* Test data 2 of test case 3 *)
  END_VAR

                    (*Run the test cases*)
TEST_CASE_1_SETUP();
TEST_CASE_1_EXEC();

TEST_CASE_2_SETUP();
TEST_CASE_2_EXEC();

TEST_CASE_3_SETUP();
TEST_CASE_3_EXEC();

(*Instantiate the test runner*)
testRunner(
	Id := 134,
	Name := 'assertLessEqual_DATE_AND_TIME',
    RunTests := GVL.RunAll OR vRunAll,
	ResetTests := GVL.ResetAll OR vResetAll,
	TestCases:=vTestCases);

(*Report the results to the collection global*)
GVL.Results[testRunner.Id] := testRunner.Summary;
                  

ACTION TEST_CASE_1_SETUP:
                        IF vTestCases[0].state = utTestCaseStates.ut_SETUP THEN
	(*Setup the test case information*)
	vTestCases[0].id := 1;
	vTestCases[0].desc[0] := 'RETURNS TRUE WHEN PARAMETER ACT LESS THAN XP';
    vTestCases[0].desc[1] := 'Tests if the function returns True if the parameter act is less than parameter xp';
	vTestCases[0].desc[2] := 'PASS IF: Return value is TRUE';
	
	(*Setup needed variables*)
	vTestCase1_act := REAL_TO_DT(85.4);
	vTestCase1_xp := REAL_TO_DT(115.4);
END_IF
                      
END_ACTION

ACTION TEST_CASE_3_SETUP:
                        IF vTestCases[2].state = utTestCaseStates.ut_SETUP THEN
	(*Setup the test case information*)
	vTestCases[2].id := 3;
    vTestCases[2].desc[0] := 'RETURNS FALSE WHEN PARAMETER ACT GREATER THAN XP';
    vTestCases[2].desc[1] := 'Tests if the function returns False if the parameter act is greater than parameter xp';
	vTestCases[2].desc[2] := 'PASS IF: Return value is FALSE';
	
	(*Setup needed variables*)
	vTestCase3_act := REAL_TO_DT(115.4);
	vTestCase3_xp := REAL_TO_DT(85.4);
END_IF
                      
END_ACTION

ACTION TEST_CASE_3_EXEC:
                        IF vTestCases[2].state = utTestCaseStates.ut_RUNNING THEN
	(*Run the test case*)
	IF NOT assertLessEqual_DATE_AND_TIME(vTestCase3_act, vTestCase3_xp) THEN
		vTestCases[2].state := utTestCaseStates.ut_PASSED;
		vTestCases[2].msg := 'Parameter act was greater than xp and function returned FALSE -> PASS';
	ELSE
		vTestCases[2].state := utTestCaseStates.ut_FAILED;
		vTestCases[2].msg := 'Parameter act was greater than xp and function returned TRUE -> FAIL';
	END_IF
END_IF
                      
END_ACTION

ACTION TEST_CASE_1_EXEC:
                        IF vTestCases[0].state = utTestCaseStates.ut_RUNNING THEN
	(*Run the test case*)
	IF assertLessEqual_DATE_AND_TIME(vTestCase1_act, vTestCase1_xp) THEN
		vTestCases[0].state := utTestCaseStates.ut_PASSED;
		vTestCases[0].msg := 'Parameter act was less than xp and function returned TRUE -> PASS';
	ELSE
		vTestCases[0].state := utTestCaseStates.ut_FAILED;
		vTestCases[0].msg := 'Parameter act was less than xp and function returned FALSE -> FAIL';
	END_IF
END_IF
                      
END_ACTION

ACTION TEST_CASE_2_SETUP:
                        IF vTestCases[1].state = utTestCaseStates.ut_SETUP THEN
	(*Setup the test case information*)
	vTestCases[1].id := 2;
    vTestCases[1].desc[0] := 'RETURNS TRUE WHEN PARAMETER ACT EQUAL TO XP';
    vTestCases[1].desc[1] := 'Tests if the function returns True if the parameter act is equal to parameter xp';
	vTestCases[1].desc[2] := 'PASS IF: Return value is TRUE';
	
	(*Setup needed variables*)
	vTestCase2_act := REAL_TO_DT(115.4);
	vTestCase2_xp := REAL_TO_DT(115.4);
END_IF
                      
END_ACTION

ACTION TEST_CASE_2_EXEC:
                        IF vTestCases[1].state = utTestCaseStates.ut_RUNNING THEN
	(*Run the test case*)
	IF assertLessEqual_DATE_AND_TIME(vTestCase2_act, vTestCase2_xp) THEN
		vTestCases[1].state := utTestCaseStates.ut_PASSED;
		vTestCases[1].msg := 'Parameter act was equal to xp and function returned TRUE -> PASS';
	ELSE
		vTestCases[1].state := utTestCaseStates.ut_FAILED;
		vTestCases[1].msg := 'Parameter act was equal to xp and function returned FALSE -> FAIL';
	END_IF
END_IF
                      
END_ACTION
END_PROGRAM

PROGRAM test_assertArrayEqual_UINT
  VAR
    vTestCases : ARRAY[0..20] OF utTestCase;  (* Definition of all test cases for this POU *)
    testRunner : utTestSuite;  (* Test Suite fb instance to run the tests *)
    vRunAll : BOOL;  (* Manual command to run all tests for this POU *)
    vResetAll : BOOL;  (* Manual command to reset all tests for this POU *)
    vTestCase1_act : ARRAY[0..70] OF UINT;  (* Array data 1 of test case 1 *)
    vTestCase1_xp : ARRAY[0..70] OF UINT;  (* Array data 2 of test case 1 *)
    vTestCase2_act : ARRAY[0..70] OF UINT;  (* Array data 3 of test case 2 *)
    vTestCase2_xp : ARRAY[0..70] OF UINT;  (* Array data 4 of test case 2 *)
    i : UINT;  (* Iterator variable i *)
    j : UINT;  (* Iterator variable j *)
  END_VAR

                    (*Run the test cases*)
TEST_CASE_1_SETUP();
TEST_CASE_1_EXEC();

TEST_CASE_2_SETUP();
TEST_CASE_2_EXEC();

(*Instantiate the test runner*)
testRunner(
	Id := 146,
	Name := 'assertArrayEqual_UINT',
    RunTests := GVL.RunAll OR vRunAll,
	ResetTests := GVL.ResetAll OR vResetAll,
	TestCases:=vTestCases);

(*Report the results to the collection global*)
GVL.Results[testRunner.Id] := testRunner.Summary;
                  

ACTION TEST_CASE_2_EXEC:
                        IF vTestCases[1].state = utTestCaseStates.ut_RUNNING THEN
	(*Run the test case*)
	IF NOT assertArrayEqual_UINT(ADR(vTestCase2_act), ADR(vTestCase2_xp), SIZEOF(vTestCase2_act)) THEN
		vTestCases[1].state := utTestCaseStates.ut_PASSED;
		vTestCases[1].msg := 'Arrays were not equal and function returned FALSE -> PASS';
	ELSE
		vTestCases[1].state := utTestCaseStates.ut_FAILED;
		vTestCases[1].msg := 'Arrays were not equal and function returned TRUE -> FAIL';
	END_IF
END_IF
                      
END_ACTION

ACTION TEST_CASE_1_SETUP:
                        IF vTestCases[0].state = utTestCaseStates.ut_SETUP THEN
	(*Setup the test case information*)
	vTestCases[0].id := 1;
	vTestCases[0].desc[0] := 'RETURNS TRUE WHEN ARRAYS EQUAL';
    vTestCases[0].desc[1] := 'Tests if the function returns True if the passed in arrays are identical';
	vTestCases[0].desc[2] := 'PASS IF: Return value is TRUE';
	
	(*Setup needed variables*)
	FOR i:=0 TO 70 DO
		vTestCase1_act[i] := 35 * BOOL_TO_UINT(i MOD 2 = 0);
		vTestCase1_xp[i] := 35 * BOOL_TO_UINT(i MOD 2 = 0);
	END_FOR
END_IF
                      
END_ACTION

ACTION TEST_CASE_1_EXEC:
                        IF vTestCases[0].state = utTestCaseStates.ut_RUNNING THEN
	(*Run the test case*)
	IF assertArrayEqual_UINT(ADR(vTestCase1_act), ADR(vTestCase1_xp), SIZEOF(vTestCase1_act)) THEN
		vTestCases[0].state := utTestCaseStates.ut_PASSED;
		vTestCases[0].msg := 'Arrays were equal and function returned TRUE -> PASS';
	ELSE
		vTestCases[0].state := utTestCaseStates.ut_FAILED;
		vTestCases[0].msg := 'Arrays were equal and function returned FALSE -> FAIL';
	END_IF
END_IF
                      
END_ACTION

ACTION TEST_CASE_2_SETUP:
                        IF vTestCases[1].state = utTestCaseStates.ut_SETUP THEN
	(*Setup the test case information*)
	vTestCases[1].id := 2;
	vTestCases[1].desc[0] := 'RETURNS FALSE WHEN ARRAYS NOT EQUAL';
    vTestCases[1].desc[1] := 'Tests if the function returns False if the passed in arrays are not identical';
	vTestCases[1].desc[2] := 'PASS IF: Return value is FALSE';
	
	(*Setup needed variables*)
	FOR j:=0 TO 70 DO
		vTestCase2_act[j] := 35 * BOOL_TO_UINT(j MOD 2 = 0);
		vTestCase2_xp[j] := 35 * BOOL_TO_UINT(j MOD 2 <> 0);
	END_FOR
END_IF
                      
END_ACTION
END_PROGRAM

PROGRAM test_assertArrayEqual_BYTE
  VAR
    vTestCases : ARRAY[0..20] OF utTestCase;  (* Definition of all test cases for this POU *)
    testRunner : utTestSuite;  (* Test Suite fb instance to run the tests *)
    vRunAll : BOOL;  (* Manual command to run all tests for this POU *)
    vResetAll : BOOL;  (* Manual command to reset all tests for this POU *)
    vTestCase1_act : ARRAY[0..70] OF BYTE;  (* Array data 1 of test case 1 *)
    vTestCase1_xp : ARRAY[0..70] OF BYTE;  (* Array data 2 of test case 1 *)
    vTestCase2_act : ARRAY[0..70] OF BYTE;  (* Array data 3 of test case 2 *)
    vTestCase2_xp : ARRAY[0..70] OF BYTE;  (* Array data 4 of test case 2 *)
    i : UINT;  (* Iterator variable i *)
    j : UINT;  (* Iterator variable j *)
  END_VAR

                    (*Run the test cases*)
TEST_CASE_1_SETUP();
TEST_CASE_1_EXEC();

TEST_CASE_2_SETUP();
TEST_CASE_2_EXEC();

(*Instantiate the test runner*)
testRunner(
	Id := 139,
	Name := 'assertArrayEqual_BYTE',
    RunTests := GVL.RunAll OR vRunAll,
	ResetTests := GVL.ResetAll OR vResetAll,
	TestCases:=vTestCases);

(*Report the results to the collection global*)
GVL.Results[testRunner.Id] := testRunner.Summary;
                  

ACTION TEST_CASE_2_EXEC:
                        IF vTestCases[1].state = utTestCaseStates.ut_RUNNING THEN
	(*Run the test case*)
	IF NOT assertArrayEqual_BYTE(ADR(vTestCase2_act), ADR(vTestCase2_xp), SIZEOF(vTestCase2_act)) THEN
		vTestCases[1].state := utTestCaseStates.ut_PASSED;
		vTestCases[1].msg := 'Arrays were not equal and function returned FALSE -> PASS';
	ELSE
		vTestCases[1].state := utTestCaseStates.ut_FAILED;
		vTestCases[1].msg := 'Arrays were not equal and function returned TRUE -> FAIL';
	END_IF
END_IF
                      
END_ACTION

ACTION TEST_CASE_1_SETUP:
                        IF vTestCases[0].state = utTestCaseStates.ut_SETUP THEN
	(*Setup the test case information*)
	vTestCases[0].id := 1;
	vTestCases[0].desc[0] := 'RETURNS TRUE WHEN ARRAYS EQUAL';
    vTestCases[0].desc[1] := 'Tests if the function returns True if the passed in arrays are identical';
	vTestCases[0].desc[2] := 'PASS IF: Return value is TRUE';
	
	(*Setup needed variables*)
	FOR i:=0 TO 70 DO
		vTestCase1_act[i] := UINT_TO_BYTE(35 * BOOL_TO_UINT(i MOD 2 = 0));
		vTestCase1_xp[i] := UINT_TO_BYTE(35 * BOOL_TO_UINT(i MOD 2 = 0));
	END_FOR
END_IF
                      
END_ACTION

ACTION TEST_CASE_1_EXEC:
                        IF vTestCases[0].state = utTestCaseStates.ut_RUNNING THEN
	(*Run the test case*)
	IF assertArrayEqual_BYTE(ADR(vTestCase1_act), ADR(vTestCase1_xp), SIZEOF(vTestCase1_act)) THEN
		vTestCases[0].state := utTestCaseStates.ut_PASSED;
		vTestCases[0].msg := 'Arrays were equal and function returned TRUE -> PASS';
	ELSE
		vTestCases[0].state := utTestCaseStates.ut_FAILED;
		vTestCases[0].msg := 'Arrays were equal and function returned FALSE -> FAIL';
	END_IF
END_IF
                      
END_ACTION

ACTION TEST_CASE_2_SETUP:
                        IF vTestCases[1].state = utTestCaseStates.ut_SETUP THEN
	(*Setup the test case information*)
	vTestCases[1].id := 2;
	vTestCases[1].desc[0] := 'RETURNS FALSE WHEN ARRAYS NOT EQUAL';
    vTestCases[1].desc[1] := 'Tests if the function returns False if the passed in arrays are not identical';
	vTestCases[1].desc[2] := 'PASS IF: Return value is FALSE';
	
	(*Setup needed variables*)
	FOR j:=0 TO 70 DO
		vTestCase2_act[j] := UINT_TO_BYTE(35 * BOOL_TO_UINT(j MOD 2 = 0));
		vTestCase2_xp[j] := UINT_TO_BYTE(35 * BOOL_TO_UINT(j MOD 2 <> 0));
	END_FOR
END_IF
                      
END_ACTION
END_PROGRAM

PROGRAM test_assertEqual_BYTE
  VAR
    vTestCases : ARRAY[0..20] OF utTestCase;  (* Definition of all test cases for this POU *)
    testRunner : utTestSuite;  (* Test Suite fb instance to run the tests *)
    vRunAll : BOOL;  (* Manual command to run all tests for this POU *)
    vResetAll : BOOL;  (* Manual command to reset all tests for this POU *)
    vTestCase1_act : BYTE;  (* Test data 1 of test case 1 *)
    vTestCase1_xp : BYTE;  (* Test data 2 of test case 1 *)
    vTestCase2_act : BYTE;  (* Test data 1 of test case 2 *)
    vTestCase2_xp : BYTE;  (* Test data 2 of test case 2 *)
  END_VAR

                    (*Run the test cases*)
TEST_CASE_1_SETUP();
TEST_CASE_1_EXEC();

TEST_CASE_2_SETUP();
TEST_CASE_2_EXEC();

(*Instantiate the test runner*)
testRunner(
	Id := 1,
	Name := 'assertEqual_BYTE',
    RunTests := GVL.RunAll OR vRunAll,
	ResetTests := GVL.ResetAll OR vResetAll,
	TestCases:=vTestCases);

(*Report the results to the collection global*)
GVL.Results[testRunner.Id] := testRunner.Summary;
                  

ACTION TEST_CASE_1_EXEC:
                        IF vTestCases[0].state = utTestCaseStates.ut_RUNNING THEN
	(*Run the test case*)
	IF assertEqual_BYTE(vTestCase1_act, vTestCase1_xp) THEN
		vTestCases[0].state := utTestCaseStates.ut_PASSED;
		vTestCases[0].msg := 'Passed parameters were equal and function returned TRUE -> PASS';
	ELSE
		vTestCases[0].state := utTestCaseStates.ut_FAILED;
		vTestCases[0].msg := 'Passed parameters were equal and function returned FALSE -> FAIL';
	END_IF
END_IF
                      
END_ACTION

ACTION TEST_CASE_1_SETUP:
                        IF vTestCases[0].state = utTestCaseStates.ut_SETUP THEN
	(*Setup the test case information*)
	vTestCases[0].id := 1;
	vTestCases[0].desc[0] := 'RETURNS TRUE WHEN PARAMETERS EQUAL';
    vTestCases[0].desc[1] := 'Tests if the function returns True if the passed in parameters hold the same value';
	vTestCases[0].desc[2] := 'PASS IF: Return value is TRUE';
	
	(*Setup needed variables*)
	vTestCase1_act := REAL_TO_BYTE(115.4);
	vTestCase1_xp := REAL_TO_BYTE(115.4);
END_IF
                      
END_ACTION

ACTION TEST_CASE_2_SETUP:
                        IF vTestCases[1].state = utTestCaseStates.ut_SETUP THEN
	(*Setup the test case information*)
	vTestCases[1].id := 2;
	vTestCases[1].desc[0] := 'RETURNS FALSE WHEN PARAMETERS NOT EQUAL';
    vTestCases[1].desc[1] := 'Tests if the function returns False if the passed in parameters do not hold the same value';
	vTestCases[1].desc[2] := 'PASS IF: Return value is FALSE';
	
	(*Setup needed variables*)
	vTestCase2_act := REAL_TO_BYTE(115.4);
	vTestCase2_xp := REAL_TO_BYTE(-84.4);
END_IF
                      
END_ACTION

ACTION TEST_CASE_2_EXEC:
                        IF vTestCases[1].state = utTestCaseStates.ut_RUNNING THEN
	(*Run the test case*)
	IF NOT assertEqual_BYTE(vTestCase2_act, vTestCase2_xp) THEN
		vTestCases[1].state := utTestCaseStates.ut_PASSED;
		vTestCases[1].msg := 'Passed parameters were not equal and function returned FALSE -> PASS';
	ELSE
		vTestCases[1].state := utTestCaseStates.ut_FAILED;
		vTestCases[1].msg := 'Passed parameters were not equal and function returned TRUE -> FAIL';
	END_IF
END_IF
                      
END_ACTION
END_PROGRAM

PROGRAM test_assertEqual_TIME_OF_DAY
  VAR
    vTestCases : ARRAY[0..20] OF utTestCase;  (* Definition of all test cases for this POU *)
    testRunner : utTestSuite;  (* Test Suite fb instance to run the tests *)
    vRunAll : BOOL;  (* Manual command to run all tests for this POU *)
    vResetAll : BOOL;  (* Manual command to reset all tests for this POU *)
    vTestCase1_act : TOD;  (* Test data 1 of test case 1 *)
    vTestCase1_xp : TOD;  (* Test data 2 of test case 1 *)
    vTestCase2_act : TOD;  (* Test data 1 of test case 2 *)
    vTestCase2_xp : TOD;  (* Test data 2 of test case 2 *)
  END_VAR

                    (*Run the test cases*)
TEST_CASE_1_SETUP();
TEST_CASE_1_EXEC();

TEST_CASE_2_SETUP();
TEST_CASE_2_EXEC();

(*Instantiate the test runner*)
testRunner(
	Id := 23,
	Name := 'assertEqual_TIME_OF_DAY',
    RunTests := GVL.RunAll OR vRunAll,
	ResetTests := GVL.ResetAll OR vResetAll,
	TestCases:=vTestCases);

(*Report the results to the collection global*)
GVL.Results[testRunner.Id] := testRunner.Summary;
                  

ACTION TEST_CASE_2_EXEC:
                        IF vTestCases[1].state = utTestCaseStates.ut_RUNNING THEN
	(*Run the test case*)
	IF NOT assertEqual_TIME_OF_DAY(vTestCase2_act, vTestCase2_xp) THEN
		vTestCases[1].state := utTestCaseStates.ut_PASSED;
		vTestCases[1].msg := 'Passed parameters were not equal and function returned FALSE -> PASS';
	ELSE
		vTestCases[1].state := utTestCaseStates.ut_FAILED;
		vTestCases[1].msg := 'Passed parameters were not equal and function returned TRUE -> FAIL';
	END_IF
END_IF
                      
END_ACTION

ACTION TEST_CASE_1_SETUP:
                        IF vTestCases[0].state = utTestCaseStates.ut_SETUP THEN
	(*Setup the test case information*)
	vTestCases[0].id := 1;
	vTestCases[0].desc[0] := 'RETURNS TRUE WHEN PARAMETERS EQUAL';
    vTestCases[0].desc[1] := 'Tests if the function returns True if the passed in parameters hold the same value';
	vTestCases[0].desc[2] := 'PASS IF: Return value is TRUE';
	
	(*Setup needed variables*)
	vTestCase1_act := REAL_TO_TOD(115.4);
	vTestCase1_xp := REAL_TO_TOD(115.4);
END_IF
                      
END_ACTION

ACTION TEST_CASE_1_EXEC:
                        IF vTestCases[0].state = utTestCaseStates.ut_RUNNING THEN
	(*Run the test case*)
	IF assertEqual_TIME_OF_DAY(vTestCase1_act, vTestCase1_xp) THEN
		vTestCases[0].state := utTestCaseStates.ut_PASSED;
		vTestCases[0].msg := 'Passed parameters were equal and function returned TRUE -> PASS';
	ELSE
		vTestCases[0].state := utTestCaseStates.ut_FAILED;
		vTestCases[0].msg := 'Passed parameters were equal and function returned FALSE -> FAIL';
	END_IF
END_IF
                      
END_ACTION

ACTION TEST_CASE_2_SETUP:
                        IF vTestCases[1].state = utTestCaseStates.ut_SETUP THEN
	(*Setup the test case information*)
	vTestCases[1].id := 2;
	vTestCases[1].desc[0] := 'RETURNS FALSE WHEN PARAMETERS NOT EQUAL';
    vTestCases[1].desc[1] := 'Tests if the function returns False if the passed in parameters do not hold the same value';
	vTestCases[1].desc[2] := 'PASS IF: Return value is FALSE';
	
	(*Setup needed variables*)
	vTestCase2_act := REAL_TO_TOD(115.4);
	vTestCase2_xp := REAL_TO_TOD(-84.4);
END_IF
                      
